LIN {X 0,Y 412.801,Z 579.645,A -85,B 0,C 180,E1 -10545.301,E2 -10545.301} C_VEL
LIN {X 0,Y 413.785,Z 567.872,A -85,B 0,C 180,E1 -10546.655,E2 -10546.655} C_VEL
LIN {X 0,Y 414.83,Z 556.165,A -85,B 0,C 180,E1 -10547.755,E2 -10547.755} C_VEL
LIN {X 0,Y 415.847,Z 543.386,A -85,B 0,C 180,E1 -10548.73,E2 -10548.73} C_VEL
LIN {X 0,Y 416.624,Z 531.359,A -85,B 0,C 180,E1 -10549.46,E2 -10549.46} C_VEL
LIN {X 0,Y 414.513,Z 516.688,A -85,B 0,C 180,E1 -10550.265,E2 -10550.265} C_VEL
LIN {X 0,Y 411.69,Z 501.521,A -85,B 0,C 180,E1 -10550.902,E2 -10550.902} C_VEL
LIN {X 0,Y 410.791,Z 496.633,A -85,B 0,C 180,E1 -10551.088,E2 -10551.088} C_VEL
LIN {X 0,Y 411.227,Z 488.281,A -85,B 0,C 180,E1 -10554.65,E2 -10554.65} C_VEL
LIN {X 0,Y 411.681,Z 480.635,A -85,B 0,C 180,E1 -10557.999,E2 -10557.999} C_VEL
LIN {X 0,Y 412.119,Z 474.429,A -85,B 0,C 180,E1 -10560.77,E2 -10560.77} C_VEL
LIN {X 0,Y 412.63,Z 468.653,A -85,B 0,C 180,E1 -10563.428,E2 -10563.428} C_VEL
LIN {X 0,Y 413.208,Z 461.279,A -85,B 0,C 180,E1 -10566.928,E2 -10566.928} C_VEL
LIN {X 0,Y 413.477,Z 457.145,A -85,B 0,C 180,E1 -10568.968,E2 -10568.968} C_VEL
LIN {X 0,Y 412.933,Z 452.303,A -85,B 0,C 180,E1 -10571.508,E2 -10571.508} C_VEL
LIN {X 0,Y 411.832,Z 446.077,A -85,B 0,C 180,E1 -10574.979,E2 -10574.979} C_VEL
LIN {X 0,Y 411.236,Z 442.884,A -85,B 0,C 180,E1 -10576.875,E2 -10576.875} C_VEL
LIN {X 0,Y 411.214,Z 442.889,A -85,B 0,C 180,E1 -10580.271,E2 -10580.271} C_VEL
LIN {X 0,Y 411.188,Z 442.891,A -85,B 0,C 180,E1 -10583.447,E2 -10583.447} C_VEL
LIN {X 0,Y 411.203,Z 442.89,A -85,B 0,C 180,E1 -10586.873,E2 -10586.873} C_VEL
LIN {X 0,Y 411.236,Z 442.886,A -85,B 0,C 180,E1 -10590.642,E2 -10590.642} C_VEL
LIN {X 0,Y 411.233,Z 442.885,A -85,B 0,C 180,E1 -10593.619,E2 -10593.619} C_VEL
LIN {X 0,Y 411.197,Z 442.892,A -85,B 0,C 180,E1 -10596.852,E2 -10596.852} C_VEL
LIN {X 0,Y 411.209,Z 442.888,A -85,B 0,C 180,E1 -10600.05,E2 -10600.05} C_VEL
LIN {X 0,Y 411.257,Z 442.883,A -85,B 0,C 180,E1 -10603.131,E2 -10603.131} C_VEL
LIN {X 0,Y 411.299,Z 442.879,A -85,B 0,C 180,E1 -10606.896,E2 -10606.896} C_VEL
LIN {X 0,Y 411.288,Z 442.878,A -85,B 0,C 180,E1 -10610.161,E2 -10610.161} C_VEL
LIN {X 0,Y 411.454,Z 442.859,A -85,B 0,C 180,E1 -10613.133,E2 -10613.133} C_VEL
LIN {X 0,Y 411.307,Z 442.876,A -85,B 0,C 180,E1 -10615.099,E2 -10615.099} C_VEL
LIN {X 0,Y 411.508,Z 442.851,A -85,B 0,C 180,E1 -10618.043,E2 -10618.043} C_VEL
LIN {X 0,Y 411.635,Z 442.834,A -85,B 0,C 180,E1 -10620,E2 -10620} C_VEL
LIN {X 0,Y 411.462,Z 442.858,A -85,B 0,C 180,E1 -10622.937,E2 -10622.937} C_VEL
LIN {X 0,Y 411.453,Z 442.858,A -85,B 0,C 180,E1 -10626.597,E2 -10626.597} C_VEL
LIN {X 0,Y 411.348,Z 442.871,A -85,B 0,C 180,E1 -10628.846,E2 -10628.846} C_VEL
LIN {X 0,Y 411.278,Z 442.88,A -85,B 0,C 180,E1 -10631.833,E2 -10631.833} C_VEL
LIN {X 0,Y 411.254,Z 442.884,A -85,B 0,C 180,E1 -10634.853,E2 -10634.853} C_VEL
LIN {X 0,Y 411.247,Z 442.883,A -85,B 0,C 180,E1 -10637.916,E2 -10637.916} C_VEL
LIN {X 0,Y 411.191,Z 442.89,A -85,B 0,C 180,E1 -10641.035,E2 -10641.035} C_VEL
LIN {X 0,Y 411.223,Z 442.888,A -85,B 0,C 180,E1 -10644.216,E2 -10644.216} C_VEL
LIN {X 0,Y 411.254,Z 442.881,A -85,B 0,C 180,E1 -10647.478,E2 -10647.478} C_VEL
LIN {X 0,Y 411.185,Z 442.89,A -85,B 0,C 180,E1 -10650.848,E2 -10650.848} C_VEL
LIN {X 0,Y 411.203,Z 442.891,A -85,B 0,C 180,E1 -10654.334,E2 -10654.334} C_VEL
LIN {X 0,Y 411.196,Z 442.892,A -85,B 0,C 180,E1 -10657.974,E2 -10657.974} C_VEL
LIN {X 0,Y 411.162,Z 442.892,A -85,B 0,C 180,E1 -10661.229,E2 -10661.229} C_VEL
LIN {X 0,Y 411.178,Z 442.892,A -85,B 0,C 180,E1 -10664.491,E2 -10664.491} C_VEL
LIN {X 0,Y 411.197,Z 442.892,A -85,B 0,C 180,E1 -10668.198,E2 -10668.198} C_VEL
LIN {X 0,Y 411.23,Z 442.885,A -85,B 0,C 180,E1 -10670.778,E2 -10670.778} C_VEL
LIN {X 0,Y 411.2,Z 442.889,A -85,B 0,C 180,E1 -10674.472,E2 -10674.472} C_VEL
LIN {X 0,Y 411.208,Z 442.887,A -85,B 0,C 180,E1 -10676.874,E2 -10676.874} C_VEL
LIN {X 0,Y 411.242,Z 442.883,A -85,B 0,C 180,E1 -10680.643,E2 -10680.643} C_VEL
LIN {X 0,Y 411.24,Z 442.887,A -85,B 0,C 180,E1 -10683.62,E2 -10683.62} C_VEL
LIN {X 0,Y 411.206,Z 442.887,A -85,B 0,C 180,E1 -10686.853,E2 -10686.853} C_VEL
LIN {X 0,Y 411.218,Z 442.889,A -85,B 0,C 180,E1 -10690.051,E2 -10690.051} C_VEL
LIN {X 0,Y 411.266,Z 442.881,A -85,B 0,C 180,E1 -10693.132,E2 -10693.132} C_VEL
LIN {X 0,Y 411.309,Z 442.874,A -85,B 0,C 180,E1 -10696.896,E2 -10696.896} C_VEL
LIN {X 0,Y 411.296,Z 442.877,A -85,B 0,C 180,E1 -10700.162,E2 -10700.162} C_VEL
LIN {X 0,Y 411.427,Z 442.863,A -85,B 0,C 180,E1 -10703.133,E2 -10703.133} C_VEL
LIN {X 0,Y 411.31,Z 442.876,A -85,B 0,C 180,E1 -10705.099,E2 -10705.099} C_VEL
LIN {X 0,Y 411.518,Z 442.85,A -85,B 0,C 180,E1 -10708.043,E2 -10708.043} C_VEL
LIN {X 0,Y 411.644,Z 442.833,A -85,B 0,C 180,E1 -10710,E2 -10710} C_VEL
LIN {X 0,Y 411.462,Z 442.858,A -85,B 0,C 180,E1 -10712.937,E2 -10712.937} C_VEL
LIN {X 0,Y 411.475,Z 442.855,A -85,B 0,C 180,E1 -10715.882,E2 -10715.882} C_VEL
LIN {X 0,Y 411.355,Z 442.87,A -85,B 0,C 180,E1 -10718.845,E2 -10718.845} C_VEL
LIN {X 0,Y 411.288,Z 442.879,A -85,B 0,C 180,E1 -10721.832,E2 -10721.832} C_VEL
LIN {X 0,Y 411.263,Z 442.883,A -85,B 0,C 180,E1 -10724.852,E2 -10724.852} C_VEL
LIN {X 0,Y 411.243,Z 442.881,A -85,B 0,C 180,E1 -10727.596,E2 -10727.596} C_VEL
LIN {X 0,Y 410.583,Z 442.965,A -85,B 0,C 180,E1 -10728.414,E2 -10728.414} C_VEL
LIN {X 0,Y 407.695,Z 443.326,A -85,B 0,C 180,E1 -10729.742,E2 -10729.742} C_VEL
LIN {X 0,Y 405.25,Z 443.632,A -85,B 0,C 180,E1 -10730.814,E2 -10730.814} C_VEL
LIN {X 0,Y 404.215,Z 443.76,A -85,B 0,C 180,E1 -10731.644,E2 -10731.644} C_VEL
LIN {X 0,Y 404.139,Z 443.767,A -85,B 0,C 180,E1 -10731.926,E2 -10731.926} C_VEL
LIN {X 0,Y 404.218,Z 443.761,A -85,B 0,C 180,E1 -10735.296,E2 -10735.296} C_VEL
LIN {X 0,Y 404.197,Z 443.76,A -85,B 0,C 180,E1 -10737.999,E2 -10737.999} C_VEL
LIN {X 0,Y 404.138,Z 443.768,A -85,B 0,C 180,E1 -10741.557,E2 -10741.557} C_VEL
LIN {X 0,Y 404.105,Z 443.772,A -85,B 0,C 180,E1 -10743.815,E2 -10743.815} C_VEL
LIN {X 0,Y 403.874,Z 443.805,A -85,B 0,C 180,E1 -10746.825,E2 -10746.825} C_VEL
LIN {X 0,Y 403.436,Z 443.861,A -85,B 0,C 180,E1 -10750.131,E2 -10750.131} C_VEL
LIN {X 0,Y 403.357,Z 444.539,A -85,B 0,C 180,E1 -10751.476,E2 -10751.476} C_VEL
LIN {X 0,Y 403.264,Z 447.096,A -85,B 0,C 180,E1 -10754.394,E2 -10754.394} C_VEL
LIN {X 0,Y 403.237,Z 449.596,A -85,B 0,C 180,E1 -10757.177,E2 -10757.177} C_VEL
LIN {X 0,Y 403.147,Z 452.843,A -85,B 0,C 180,E1 -10760.723,E2 -10760.723} C_VEL
LIN {X 0,Y 407.346,Z 467.682,A -85,B 0,C 180,E1 -10761.418,E2 -10761.418} C_VEL
LIN {X 0,Y 410.494,Z 480.117,A -85,B 0,C 180,E1 -10762.156,E2 -10762.156} C_VEL
LIN {X 0,Y 409.792,Z 493.988,A -85,B 0,C 180,E1 -10762.977,E2 -10762.977} C_VEL
LIN {X 0,Y 408.853,Z 507.194,A -85,B 0,C 180,E1 -10763.977,E2 -10763.977} C_VEL
LIN {X 0,Y 407.914,Z 518.652,A -85,B 0,C 180,E1 -10765.049,E2 -10765.049} C_VEL
LIN {X 0,Y 406.818,Z 530.774,A -85,B 0,C 180,E1 -10766.439,E2 -10766.439} C_VEL
LIN {X 0,Y 405.964,Z 540.883,A -85,B 0,C 180,E1 -10767.852,E2 -10767.852} C_VEL
LIN {X 0,Y 405.008,Z 550.623,A -85,B 0,C 180,E1 -10769.498,E2 -10769.498} C_VEL
LIN {X 0,Y 404.378,Z 558.657,A -85,B 0,C 180,E1 -10771.165,E2 -10771.165} C_VEL
LIN {X 0,Y 403.791,Z 566.103,A -85,B 0,C 180,E1 -10773.093,E2 -10773.093} C_VEL
LIN {X 0,Y 403.401,Z 571.667,A -85,B 0,C 180,E1 -10774.948,E2 -10774.948} C_VEL
LIN {X 0,Y 403.096,Z 576.05,A -85,B 0,C 180,E1 -10776.903,E2 -10776.903} C_VEL
LIN {X 0,Y 402.928,Z 578.626,A -85,B 0,C 180,E1 -10778.513,E2 -10778.513} C_VEL
LIN {X 0,Y 402.891,Z 580.598,A -85,B 0,C 180,E1 -10780.644,E2 -10780.644} C_VEL
LIN {X 0,Y 402.812,Z 581.067,A -85,B 0,C 180,E1 -10782.746,E2 -10782.746} C_VEL
LIN {X 0,Y 402.892,Z 580.745,A -85,B 0,C 180,E1 -10783.793,E2 -10783.793} C_VEL
LIN {X 0,Y 402.994,Z 579.036,A -85,B 0,C 180,E1 -10785.868,E2 -10785.868} C_VEL
LIN {X 0,Y 403.289,Z 575.854,A -85,B 0,C 180,E1 -10787.929,E2 -10787.929} C_VEL
LIN {X 0,Y 403.699,Z 571.129,A -85,B 0,C 180,E1 -10789.974,E2 -10789.974} C_VEL
LIN {X 0,Y 404.133,Z 566.55,A -85,B 0,C 180,E1 -10791.499,E2 -10791.499} C_VEL
LIN {X 0,Y 404.794,Z 559.874,A -85,B 0,C 180,E1 -10793.27,E2 -10793.27} C_VEL
LIN {X 0,Y 405.692,Z 551.582,A -85,B 0,C 180,E1 -10795.031,E2 -10795.031} C_VEL
LIN {X 0,Y 406.521,Z 543.028,A -85,B 0,C 180,E1 -10796.531,E2 -10796.531} C_VEL
LIN {X 0,Y 407.677,Z 532.688,A -85,B 0,C 180,E1 -10798.024,E2 -10798.024} C_VEL
LIN {X 0,Y 408.851,Z 521.23,A -85,B 0,C 180,E1 -10799.384,E2 -10799.384} C_VEL
LIN {X 0,Y 409.933,Z 509.849,A -85,B 0,C 180,E1 -10800.491,E2 -10800.491} C_VEL
LIN {X 0,Y 410.984,Z 497.505,A -85,B 0,C 180,E1 -10801.47,E2 -10801.47} C_VEL
LIN {X 0,Y 411.945,Z 484.382,A -85,B 0,C 180,E1 -10802.291,E2 -10802.291} C_VEL
LIN {X 0,Y 411.781,Z 481.336,A -85,B 0,C 180,E1 -10802.475,E2 -10802.475} C_VEL
LIN {X 0,Y 408.191,Z 469.01,A -85,B 0,C 180,E1 -10803.332,E2 -10803.332} C_VEL
LIN {X 0,Y 403.763,Z 456.429,A -85,B 0,C 180,E1 -10804.117,E2 -10804.117} C_VEL
LIN {X 0,Y 403.9,Z 455.086,A -85,B 0,C 180,E1 -10805.993,E2 -10805.993} C_VEL
LIN {X 0,Y 404.002,Z 453.036,A -85,B 0,C 180,E1 -10809.007,E2 -10809.007} C_VEL
LIN {X 0,Y 404.199,Z 450.477,A -85,B 0,C 180,E1 -10813.064,E2 -10813.064} C_VEL
LIN {X 0,Y 404.4,Z 448.23,A -85,B 0,C 180,E1 -10817.095,E2 -10817.095} C_VEL
LIN {X 0,Y 404.491,Z 446.675,A -85,B 0,C 180,E1 -10820.334,E2 -10820.334} C_VEL
LIN {X 0,Y 404.408,Z 445.473,A -85,B 0,C 180,E1 -10823.56,E2 -10823.56} C_VEL
LIN {X 0,Y 404.338,Z 444.649,A -85,B 0,C 180,E1 -10826.867,E2 -10826.867} C_VEL
LIN {X 0,Y 404.254,Z 444.334,A -85,B 0,C 180,E1 -10830.276,E2 -10830.276} C_VEL
LIN {X 0,Y 404.31,Z 444.687,A -85,B 0,C 180,E1 -10833.796,E2 -10833.796} C_VEL
LIN {X 0,Y 404.476,Z 445.696,A -85,B 0,C 180,E1 -10836.94,E2 -10836.94} C_VEL
LIN {X 0,Y 404.854,Z 447.496,A -85,B 0,C 180,E1 -10840.2,E2 -10840.2} C_VEL
LIN {X 0,Y 405.277,Z 449.926,A -85,B 0,C 180,E1 -10843.254,E2 -10843.254} C_VEL
LIN {X 0,Y 405.875,Z 453.507,A -85,B 0,C 180,E1 -10846.657,E2 -10846.657} C_VEL
LIN {X 0,Y 406.437,Z 457.209,A -85,B 0,C 180,E1 -10849.538,E2 -10849.538} C_VEL
LIN {X 0,Y 406.531,Z 460.16,A -85,B 0,C 180,E1 -10851.512,E2 -10851.512} C_VEL
LIN {X 0,Y 406,Z 464.25,A -85,B 0,C 180,E1 -10853.946,E2 -10853.946} C_VEL
LIN {X 0,Y 405.372,Z 469.698,A -85,B 0,C 180,E1 -10856.899,E2 -10856.899} C_VEL
LIN {X 0,Y 404.824,Z 476.312,A -85,B 0,C 180,E1 -10860.231,E2 -10860.231} C_VEL
LIN {X 0,Y 404.208,Z 483.672,A -85,B 0,C 180,E1 -10863.681,E2 -10863.681} C_VEL
LIN {X 0,Y 403.747,Z 492.25,A -85,B 0,C 180,E1 -10867.484,E2 -10867.484} C_VEL
LIN {X 0,Y 403.739,Z 493.024,A -85,B 0,C 180,E1 -10867.818,E2 -10867.818} C_VEL
LIN {X 0,Y 407.633,Z 510.63,A -85,B 0,C 180,E1 -10868.708,E2 -10868.708} C_VEL
LIN {X 0,Y 409.371,Z 523.324,A -85,B 0,C 180,E1 -10869.428,E2 -10869.428} C_VEL
LIN {X 0,Y 410.314,Z 533.68,A -85,B 0,C 180,E1 -10870.098,E2 -10870.098} C_VEL
LIN {X 0,Y 409.062,Z 547.719,A -85,B 0,C 180,E1 -10871.078,E2 -10871.078} C_VEL
LIN {X 0,Y 407.899,Z 560.436,A -85,B 0,C 180,E1 -10872.192,E2 -10872.192} C_VEL
LIN {X 0,Y 406.715,Z 572.083,A -85,B 0,C 180,E1 -10873.434,E2 -10873.434} C_VEL
LIN {X 0,Y 405.589,Z 583.695,A -85,B 0,C 180,E1 -10874.935,E2 -10874.935} C_VEL
LIN {X 0,Y 404.658,Z 593.952,A -85,B 0,C 180,E1 -10876.555,E2 -10876.555} C_VEL
LIN {X 0,Y 404.026,Z 602.53,A -85,B 0,C 180,E1 -10878.206,E2 -10878.206} C_VEL
LIN {X 0,Y 403.45,Z 610.025,A -85,B 0,C 180,E1 -10879.968,E2 -10879.968} C_VEL
LIN {X 0,Y 403.169,Z 615.304,A -85,B 0,C 180,E1 -10881.479,E2 -10881.479} C_VEL
LIN {X 0,Y 403.068,Z 619.556,A -85,B 0,C 180,E1 -10882.989,E2 -10882.989} C_VEL
LIN {X 0,Y 402.944,Z 623.879,A -85,B 0,C 180,E1 -10884.997,E2 -10884.997} C_VEL
LIN {X 0,Y 402.948,Z 626.705,A -85,B 0,C 180,E1 -10887.001,E2 -10887.001} C_VEL
LIN {X 0,Y 402.981,Z 627.576,A -85,B 0,C 180,E1 -10888.001,E2 -10888.001} C_VEL
LIN {X 0,Y 402.95,Z 628.259,A -85,B 0,C 180,E1 -10890,E2 -10890} C_VEL
LIN {X 0,Y 402.981,Z 627.549,A -85,B 0,C 180,E1 -10891.999,E2 -10891.999} C_VEL
LIN {X 0,Y 402.877,Z 625.421,A -85,B 0,C 180,E1 -10894.001,E2 -10894.001} C_VEL
LIN {X 0,Y 402.955,Z 623.822,A -85,B 0,C 180,E1 -10895.003,E2 -10895.003} C_VEL
LIN {X 0,Y 403.064,Z 619.474,A -85,B 0,C 180,E1 -10897.011,E2 -10897.011} C_VEL
LIN {X 0,Y 403.27,Z 613.496,A -85,B 0,C 180,E1 -10899.024,E2 -10899.024} C_VEL
LIN {X 0,Y 403.653,Z 606.738,A -85,B 0,C 180,E1 -10900.787,E2 -10900.787} C_VEL
LIN {X 0,Y 404.335,Z 598.312,A -85,B 0,C 180,E1 -10902.549,E2 -10902.549} C_VEL
LIN {X 0,Y 404.942,Z 589.515,A -85,B 0,C 180,E1 -10904.062,E2 -10904.062} C_VEL
LIN {X 0,Y 405.88,Z 578.894,A -85,B 0,C 180,E1 -10905.568,E2 -10905.568} C_VEL
LIN {X 0,Y 406.897,Z 567.057,A -85,B 0,C 180,E1 -10906.946,E2 -10906.946} C_VEL
LIN {X 0,Y 407.993,Z 555.275,A -85,B 0,C 180,E1 -10908.063,E2 -10908.063} C_VEL
LIN {X 0,Y 409.075,Z 542.402,A -85,B 0,C 180,E1 -10909.051,E2 -10909.051} C_VEL
LIN {X 0,Y 409.624,Z 531.3,A -85,B 0,C 180,E1 -10909.741,E2 -10909.741} C_VEL
LIN {X 0,Y 407.503,Z 516.685,A -85,B 0,C 180,E1 -10910.568,E2 -10910.568} C_VEL
LIN {X 0,Y 404.728,Z 501.456,A -85,B 0,C 180,E1 -10911.228,E2 -10911.228} C_VEL
LIN {X 0,Y 403.718,Z 496.266,A -85,B 0,C 180,E1 -10911.442,E2 -10911.442} C_VEL
LIN {X 0,Y 404.152,Z 488.877,A -85,B 0,C 180,E1 -10914.667,E2 -10914.667} C_VEL
LIN {X 0,Y 404.619,Z 481.458,A -85,B 0,C 180,E1 -10917.967,E2 -10917.967} C_VEL
LIN {X 0,Y 405.087,Z 475.295,A -85,B 0,C 180,E1 -10920.784,E2 -10920.784} C_VEL
LIN {X 0,Y 405.626,Z 469.009,A -85,B 0,C 180,E1 -10923.73,E2 -10923.73} C_VEL
LIN {X 0,Y 406.249,Z 461.72,A -85,B 0,C 180,E1 -10927.27,E2 -10927.27} C_VEL
LIN {X 0,Y 406.486,Z 458.432,A -85,B 0,C 180,E1 -10928.919,E2 -10928.919} C_VEL
LIN {X 0,Y 406.082,Z 454.284,A -85,B 0,C 180,E1 -10931.121,E2 -10931.121} C_VEL
LIN {X 0,Y 404.965,Z 448.024,A -85,B 0,C 180,E1 -10934.64,E2 -10934.64} C_VEL
LIN {X 0,Y 404.216,Z 443.758,A -85,B 0,C 180,E1 -10937.306,E2 -10937.306} C_VEL
LIN {X 0,Y 404.165,Z 443.766,A -85,B 0,C 180,E1 -10939.955,E2 -10939.955} C_VEL
LIN {X 0,Y 404.132,Z 443.772,A -85,B 0,C 180,E1 -10943.125,E2 -10943.125} C_VEL
LIN {X 0,Y 404.14,Z 443.768,A -85,B 0,C 180,E1 -10946.187,E2 -10946.187} C_VEL
LIN {X 0,Y 404.151,Z 443.767,A -85,B 0,C 180,E1 -10949.715,E2 -10949.715} C_VEL
LIN {X 0,Y 404.19,Z 443.764,A -85,B 0,C 180,E1 -10953.123,E2 -10953.123} C_VEL
LIN {X 0,Y 404.172,Z 443.766,A -85,B 0,C 180,E1 -10955.334,E2 -10955.334} C_VEL
LIN {X 0,Y 404.133,Z 443.771,A -85,B 0,C 180,E1 -10958.58,E2 -10958.58} C_VEL
LIN {X 0,Y 404.204,Z 443.758,A -85,B 0,C 180,E1 -10961.762,E2 -10961.762} C_VEL
LIN {X 0,Y 404.2,Z 443.764,A -85,B 0,C 180,E1 -10964.882,E2 -10964.882} C_VEL
LIN {X 0,Y 404.251,Z 443.754,A -85,B 0,C 180,E1 -10967.959,E2 -10967.959} C_VEL
LIN {X 0,Y 404.427,Z 443.733,A -85,B 0,C 180,E1 -10972.1,E2 -10972.1} C_VEL
LIN {X 0,Y 404.418,Z 443.734,A -85,B 0,C 180,E1 -10974.015,E2 -10974.015} C_VEL
LIN {X 0,Y 404.477,Z 443.727,A -85,B 0,C 180,E1 -10978.009,E2 -10978.009} C_VEL
LIN {X 0,Y 404.605,Z 443.71,A -85,B 0,C 180,E1 -10980,E2 -10980} C_VEL
LIN {X 0,Y 404.419,Z 443.735,A -85,B 0,C 180,E1 -10982.989,E2 -10982.989} C_VEL
LIN {X 0,Y 404.403,Z 443.735,A -85,B 0,C 180,E1 -10986.595,E2 -10986.595} C_VEL
LIN {X 0,Y 404.285,Z 443.75,A -85,B 0,C 180,E1 -10989.001,E2 -10989.001} C_VEL
LIN {X 0,Y 404.25,Z 443.756,A -85,B 0,C 180,E1 -10992.042,E2 -10992.042} C_VEL
LIN {X 0,Y 404.2,Z 443.761,A -85,B 0,C 180,E1 -10995.118,E2 -10995.118} C_VEL
LIN {X 0,Y 404.205,Z 443.763,A -85,B 0,C 180,E1 -10998.239,E2 -10998.239} C_VEL
LIN {X 0,Y 404.134,Z 443.768,A -85,B 0,C 180,E1 -11001.42,E2 -11001.42} C_VEL
LIN {X 0,Y 404.173,Z 443.766,A -85,B 0,C 180,E1 -11004.666,E2 -11004.666} C_VEL
LIN {X 0,Y 404.191,Z 443.765,A -85,B 0,C 180,E1 -11008,E2 -11008} C_VEL
LIN {X 0,Y 404.135,Z 443.768,A -85,B 0,C 180,E1 -11011.559,E2 -11011.559} C_VEL
LIN {X 0,Y 404.182,Z 443.762,A -85,B 0,C 180,E1 -11015.017,E2 -11015.017} C_VEL
LIN {X 0,Y 404.153,Z 443.767,A -85,B 0,C 180,E1 -11018.757,E2 -11018.757} C_VEL
LIN {X 0,Y 404.122,Z 443.771,A -85,B 0,C 180,E1 -11021.601,E2 -11021.601} C_VEL
LIN {X 0,Y 404.147,Z 443.767,A -85,B 0,C 180,E1 -11024.523,E2 -11024.523} C_VEL
LIN {X 0,Y 404.17,Z 443.765,A -85,B 0,C 180,E1 -11027.301,E2 -11027.301} C_VEL
LIN {X 0,Y 404.168,Z 443.768,A -85,B 0,C 180,E1 -11029.956,E2 -11029.956} C_VEL
LIN {X 0,Y 404.141,Z 443.768,A -85,B 0,C 180,E1 -11033.125,E2 -11033.125} C_VEL
LIN {X 0,Y 404.146,Z 443.77,A -85,B 0,C 180,E1 -11036.189,E2 -11036.189} C_VEL
LIN {X 0,Y 404.155,Z 443.769,A -85,B 0,C 180,E1 -11039.716,E2 -11039.716} C_VEL
LIN {X 0,Y 404.197,Z 443.76,A -85,B 0,C 180,E1 -11043.124,E2 -11043.124} C_VEL
LIN {X 0,Y 404.18,Z 443.765,A -85,B 0,C 180,E1 -11045.335,E2 -11045.335} C_VEL
LIN {X 0,Y 404.141,Z 443.767,A -85,B 0,C 180,E1 -11048.581,E2 -11048.581} C_VEL
LIN {X 0,Y 404.213,Z 443.762,A -85,B 0,C 180,E1 -11051.762,E2 -11051.762} C_VEL
LIN {X 0,Y 404.21,Z 443.76,A -85,B 0,C 180,E1 -11054.882,E2 -11054.882} C_VEL
LIN {X 0,Y 404.26,Z 443.755,A -85,B 0,C 180,E1 -11057.959,E2 -11057.959} C_VEL
LIN {X 0,Y 404.292,Z 443.749,A -85,B 0,C 180,E1 -11060.999,E2 -11060.999} C_VEL
LIN {X 0,Y 404.397,Z 443.737,A -85,B 0,C 180,E1 -11064.015,E2 -11064.015} C_VEL
LIN {X 0,Y 404.487,Z 443.726,A -85,B 0,C 180,E1 -11068.009,E2 -11068.009} C_VEL
LIN {X 0,Y 404.614,Z 443.708,A -85,B 0,C 180,E1 -11070,E2 -11070} C_VEL
LIN {X 0,Y 404.42,Z 443.735,A -85,B 0,C 180,E1 -11072.988,E2 -11072.988} C_VEL
LIN {X 0,Y 404.422,Z 443.733,A -85,B 0,C 180,E1 -11075.985,E2 -11075.985} C_VEL
LIN {X 0,Y 404.292,Z 443.751,A -85,B 0,C 180,E1 -11079.001,E2 -11079.001} C_VEL
LIN {X 0,Y 404.26,Z 443.753,A -85,B 0,C 180,E1 -11082.041,E2 -11082.041} C_VEL
LIN {X 0,Y 404.21,Z 443.762,A -85,B 0,C 180,E1 -11085.118,E2 -11085.118} C_VEL
LIN {X 0,Y 404.213,Z 443.757,A -85,B 0,C 180,E1 -11088.238,E2 -11088.238} C_VEL
LIN {X 0,Y 404.141,Z 443.77,A -85,B 0,C 180,E1 -11091.419,E2 -11091.419} C_VEL
LIN {X 0,Y 404.139,Z 443.767,A -85,B 0,C 180,E1 -11091.926,E2 -11091.926} C_VEL
LIN {X 0,Y 403.497,Z 443.851,A -85,B 0,C 180,E1 -11092.757,E2 -11092.757} C_VEL
LIN {X 0,Y 400.664,Z 444.203,A -85,B 0,C 180,E1 -11094.109,E2 -11094.109} C_VEL
LIN {X 0,Y 398.254,Z 444.504,A -85,B 0,C 180,E1 -11095.201,E2 -11095.201} C_VEL
LIN {X 0,Y 397.219,Z 444.631,A -85,B 0,C 180,E1 -11096.045,E2 -11096.045} C_VEL
LIN {X 0,Y 397.136,Z 444.639,A -85,B 0,C 180,E1 -11096.331,E2 -11096.331} C_VEL
LIN {X 0,Y 397.124,Z 444.643,A -85,B 0,C 180,E1 -11098.543,E2 -11098.543} C_VEL
LIN {X 0,Y 397.075,Z 444.646,A -85,B 0,C 180,E1 -11102.071,E2 -11102.071} C_VEL
LIN {X 0,Y 397.018,Z 444.657,A -85,B 0,C 180,E1 -11104.503,E2 -11104.503} C_VEL
LIN {X 0,Y 396.761,Z 444.69,A -85,B 0,C 180,E1 -11107.145,E2 -11107.145} C_VEL
LIN {X 0,Y 396.382,Z 444.739,A -85,B 0,C 180,E1 -11110.323,E2 -11110.323} C_VEL
LIN {X 0,Y 396.293,Z 444.863,A -85,B 0,C 180,E1 -11111.008,E2 -11111.008} C_VEL
LIN {X 0,Y 396.224,Z 447.255,A -85,B 0,C 180,E1 -11113.769,E2 -11113.769} C_VEL
LIN {X 0,Y 396.143,Z 450.68,A -85,B 0,C 180,E1 -11117.611,E2 -11117.611} C_VEL
LIN {X 0,Y 396.086,Z 453.187,A -85,B 0,C 180,E1 -11120.365,E2 -11120.365} C_VEL
LIN {X 0,Y 400.798,Z 469.92,A -85,B 0,C 180,E1 -11121.197,E2 -11121.197} C_VEL
LIN {X 0,Y 403.757,Z 481.786,A -85,B 0,C 180,E1 -11121.929,E2 -11121.929} C_VEL
LIN {X 0,Y 402.919,Z 495.445,A -85,B 0,C 180,E1 -11122.768,E2 -11122.768} C_VEL
LIN {X 0,Y 401.902,Z 508.896,A -85,B 0,C 180,E1 -11123.83,E2 -11123.83} C_VEL
LIN {X 0,Y 400.83,Z 521.361,A -85,B 0,C 180,E1 -11125.054,E2 -11125.054} C_VEL
LIN {X 0,Y 399.823,Z 532.406,A -85,B 0,C 180,E1 -11126.378,E2 -11126.378} C_VEL
LIN {X 0,Y 398.93,Z 542.406,A -85,B 0,C 180,E1 -11127.828,E2 -11127.828} C_VEL
LIN {X 0,Y 397.983,Z 551.538,A -85,B 0,C 180,E1 -11129.422,E2 -11129.422} C_VEL
LIN {X 0,Y 397.305,Z 559.75,A -85,B 0,C 180,E1 -11131.182,E2 -11131.182} C_VEL
LIN {X 0,Y 396.717,Z 567.029,A -85,B 0,C 180,E1 -11133.144,E2 -11133.144} C_VEL
LIN {X 0,Y 396.359,Z 571.943,A -85,B 0,C 180,E1 -11134.814,E2 -11134.814} C_VEL
LIN {X 0,Y 396.093,Z 575.755,A -85,B 0,C 180,E1 -11136.47,E2 -11136.47} C_VEL
LIN {X 0,Y 395.882,Z 578.512,A -85,B 0,C 180,E1 -11138.111,E2 -11138.111} C_VEL
LIN {X 0,Y 395.811,Z 580.814,A -85,B 0,C 180,E1 -11140.283,E2 -11140.283} C_VEL
LIN {X 0,Y 395.734,Z 581.534,A -85,B 0,C 180,E1 -11142.427,E2 -11142.427} C_VEL
LIN {X 0,Y 395.826,Z 580.778,A -85,B 0,C 180,E1 -11144.554,E2 -11144.554} C_VEL
LIN {X 0,Y 396.013,Z 578.587,A -85,B 0,C 180,E1 -11146.661,E2 -11146.661} C_VEL
LIN {X 0,Y 396.397,Z 574.932,A -85,B 0,C 180,E1 -11148.753,E2 -11148.753} C_VEL
LIN {X 0,Y 396.737,Z 571.155,A -85,B 0,C 180,E1 -11150.311,E2 -11150.311} C_VEL
LIN {X 0,Y 397.386,Z 564.756,A -85,B 0,C 180,E1 -11152.356,E2 -11152.356} C_VEL
LIN {X 0,Y 398.207,Z 557.496,A -85,B 0,C 180,E1 -11154.175,E2 -11154.175} C_VEL
LIN {X 0,Y 399.198,Z 548.587,A -85,B 0,C 180,E1 -11155.962,E2 -11155.962} C_VEL
LIN {X 0,Y 400.253,Z 539.312,A -85,B 0,C 180,E1 -11157.484,E2 -11157.484} C_VEL
LIN {X 0,Y 401.508,Z 528.079,A -85,B 0,C 180,E1 -11158.997,E2 -11158.997} C_VEL
LIN {X 0,Y 402.686,Z 516.727,A -85,B 0,C 180,E1 -11160.25,E2 -11160.25} C_VEL
LIN {X 0,Y 403.878,Z 504.362,A -85,B 0,C 180,E1 -11161.371,E2 -11161.371} C_VEL
LIN {X 0,Y 405.002,Z 491.224,A -85,B 0,C 180,E1 -11162.318,E2 -11162.318} C_VEL
LIN {X 0,Y 405.512,Z 484.018,A -85,B 0,C 180,E1 -11162.746,E2 -11162.746} C_VEL
LIN {X 0,Y 402.095,Z 471.959,A -85,B 0,C 180,E1 -11163.633,E2 -11163.633} C_VEL
LIN {X 0,Y 397.322,Z 458.967,A -85,B 0,C 180,E1 -11164.518,E2 -11164.518} C_VEL
LIN {X 0,Y 396.823,Z 457.011,A -85,B 0,C 180,E1 -11164.635,E2 -11164.635} C_VEL
LIN {X 0,Y 396.975,Z 454.625,A -85,B 0,C 180,E1 -11168.142,E2 -11168.142} C_VEL
LIN {X 0,Y 397.05,Z 452.67,A -85,B 0,C 180,E1 -11171.227,E2 -11171.227} C_VEL
LIN {X 0,Y 397.193,Z 450.858,A -85,B 0,C 180,E1 -11174.342,E2 -11174.342} C_VEL
LIN {X 0,Y 397.409,Z 449.208,A -85,B 0,C 180,E1 -11177.496,E2 -11177.496} C_VEL
LIN {X 0,Y 397.477,Z 447.778,A -85,B 0,C 180,E1 -11180.709,E2 -11180.709} C_VEL
LIN {X 0,Y 397.41,Z 446.679,A -85,B 0,C 180,E1 -11184,E2 -11184} C_VEL
LIN {X 0,Y 397.389,Z 445.966,A -85,B 0,C 180,E1 -11187.375,E2 -11187.375} C_VEL
LIN {X 0,Y 397.301,Z 445.823,A -85,B 0,C 180,E1 -11190.863,E2 -11190.863} C_VEL
LIN {X 0,Y 397.398,Z 446.37,A -85,B 0,C 180,E1 -11194.466,E2 -11194.466} C_VEL
LIN {X 0,Y 397.673,Z 447.853,A -85,B 0,C 180,E1 -11198.21,E2 -11198.21} C_VEL
LIN {X 0,Y 397.995,Z 449.458,A -85,B 0,C 180,E1 -11200.796,E2 -11200.796} C_VEL
LIN {X 0,Y 398.403,Z 451.845,A -85,B 0,C 180,E1 -11203.677,E2 -11203.677} C_VEL
LIN {X 0,Y 398.931,Z 454.897,A -85,B 0,C 180,E1 -11206.603,E2 -11206.603} C_VEL
LIN {X 0,Y 399.464,Z 458.385,A -85,B 0,C 180,E1 -11209.387,E2 -11209.387} C_VEL
LIN {X 0,Y 399.543,Z 460.286,A -85,B 0,C 180,E1 -11210.711,E2 -11210.711} C_VEL
LIN {X 0,Y 399.201,Z 464.294,A -85,B 0,C 180,E1 -11213.233,E2 -11213.233} C_VEL
LIN {X 0,Y 398.355,Z 470.713,A -85,B 0,C 180,E1 -11216.845,E2 -11216.845} C_VEL
LIN {X 0,Y 397.76,Z 477.543,A -85,B 0,C 180,E1 -11220.349,E2 -11220.349} C_VEL
LIN {X 0,Y 397.159,Z 484.639,A -85,B 0,C 180,E1 -11223.744,E2 -11223.744} C_VEL
LIN {X 0,Y 396.702,Z 492.515,A -85,B 0,C 180,E1 -11227.324,E2 -11227.324} C_VEL
LIN {X 0,Y 400.543,Z 508.904,A -85,B 0,C 180,E1 -11228.172,E2 -11228.172} C_VEL
LIN {X 0,Y 402.494,Z 521.599,A -85,B 0,C 180,E1 -11228.919,E2 -11228.919} C_VEL
LIN {X 0,Y 403.646,Z 533.983,A -85,B 0,C 180,E1 -11229.755,E2 -11229.755} C_VEL
LIN {X 0,Y 402.357,Z 547.67,A -85,B 0,C 180,E1 -11230.736,E2 -11230.736} C_VEL
LIN {X 0,Y 401.134,Z 560.44,A -85,B 0,C 180,E1 -11231.882,E2 -11231.882} C_VEL
LIN {X 0,Y 399.876,Z 572.007,A -85,B 0,C 180,E1 -11233.143,E2 -11233.143} C_VEL
LIN {X 0,Y 398.689,Z 583.519,A -85,B 0,C 180,E1 -11234.668,E2 -11234.668} C_VEL
LIN {X 0,Y 397.802,Z 592.833,A -85,B 0,C 180,E1 -11236.164,E2 -11236.164} C_VEL
LIN {X 0,Y 397.063,Z 601.041,A -85,B 0,C 180,E1 -11237.737,E2 -11237.737} C_VEL
LIN {X 0,Y 396.551,Z 607.729,A -85,B 0,C 180,E1 -11239.276,E2 -11239.276} C_VEL
LIN {X 0,Y 396.206,Z 613.297,A -85,B 0,C 180,E1 -11240.814,E2 -11240.814} C_VEL
LIN {X 0,Y 395.985,Z 619.202,A -85,B 0,C 180,E1 -11242.863,E2 -11242.863} C_VEL
LIN {X 0,Y 395.86,Z 623.502,A -85,B 0,C 180,E1 -11244.907,E2 -11244.907} C_VEL
LIN {X 0,Y 395.849,Z 626.3,A -85,B 0,C 180,E1 -11246.947,E2 -11246.947} C_VEL
LIN {X 0,Y 395.91,Z 627.163,A -85,B 0,C 180,E1 -11247.965,E2 -11247.965} C_VEL
LIN {X 0,Y 395.872,Z 627.831,A -85,B 0,C 180,E1 -11250,E2 -11250} C_VEL
LIN {X 0,Y 395.91,Z 627.103,A -85,B 0,C 180,E1 -11252.035,E2 -11252.035} C_VEL
LIN {X 0,Y 395.799,Z 624.952,A -85,B 0,C 180,E1 -11254.073,E2 -11254.073} C_VEL
LIN {X 0,Y 395.908,Z 621.346,A -85,B 0,C 180,E1 -11256.114,E2 -11256.114} C_VEL
LIN {X 0,Y 395.994,Z 617.614,A -85,B 0,C 180,E1 -11257.649,E2 -11257.649} C_VEL
LIN {X 0,Y 396.207,Z 612.948,A -85,B 0,C 180,E1 -11259.186,E2 -11259.186} C_VEL
LIN {X 0,Y 396.64,Z 606.145,A -85,B 0,C 180,E1 -11260.98,E2 -11260.98} C_VEL
LIN {X 0,Y 397.347,Z 597.667,A -85,B 0,C 180,E1 -11262.773,E2 -11262.773} C_VEL
LIN {X 0,Y 397.984,Z 588.82,A -85,B 0,C 180,E1 -11264.313,E2 -11264.313} C_VEL
LIN {X 0,Y 398.972,Z 578.145,A -85,B 0,C 180,E1 -11265.845,E2 -11265.845} C_VEL
LIN {X 0,Y 400.068,Z 566.248,A -85,B 0,C 180,E1 -11267.244,E2 -11267.244} C_VEL
LIN {X 0,Y 401.184,Z 554.388,A -85,B 0,C 180,E1 -11268.38,E2 -11268.38} C_VEL
LIN {X 0,Y 402.276,Z 541.378,A -85,B 0,C 180,E1 -11269.386,E2 -11269.386} C_VEL
LIN {X 0,Y 402.77,Z 532.349,A -85,B 0,C 180,E1 -11269.959,E2 -11269.959} C_VEL
LIN {X 0,Y 400.786,Z 518.378,A -85,B 0,C 180,E1 -11270.787,E2 -11270.787} C_VEL
LIN {X 0,Y 398.144,Z 503.438,A -85,B 0,C 180,E1 -11271.479,E2 -11271.479} C_VEL
LIN {X 0,Y 396.663,Z 495.998,A -85,B 0,C 180,E1 -11271.757,E2 -11271.757} C_VEL
LIN {X 0,Y 397.123,Z 488.433,A -85,B 0,C 180,E1 -11275.133,E2 -11275.133} C_VEL
LIN {X 0,Y 397.535,Z 482.407,A -85,B 0,C 180,E1 -11277.878,E2 -11277.878} C_VEL
LIN {X 0,Y 398.13,Z 474.894,A -85,B 0,C 180,E1 -11281.382,E2 -11281.382} C_VEL
LIN {X 0,Y 398.7,Z 468.75,A -85,B 0,C 180,E1 -11284.337,E2 -11284.337} C_VEL
LIN {X 0,Y 399.385,Z 461.347,A -85,B 0,C 180,E1 -11288.016,E2 -11288.016} C_VEL
LIN {X 0,Y 399.357,Z 457.634,A -85,B 0,C 180,E1 -11289.965,E2 -11289.965} C_VEL
LIN {X 0,Y 398.489,Z 452.352,A -85,B 0,C 180,E1 -11292.914,E2 -11292.914} C_VEL
LIN {X 0,Y 397.677,Z 447.555,A -85,B 0,C 180,E1 -11295.728,E2 -11295.728} C_VEL
LIN {X 0,Y 397.15,Z 444.638,A -85,B 0,C 180,E1 -11297.572,E2 -11297.572} C_VEL
LIN {X 0,Y 397.128,Z 444.644,A -85,B 0,C 180,E1 -11301.138,E2 -11301.138} C_VEL
LIN {X 0,Y 397.115,Z 444.643,A -85,B 0,C 180,E1 -11304.496,E2 -11304.496} C_VEL
LIN {X 0,Y 397.107,Z 444.642,A -85,B 0,C 180,E1 -11307.931,E2 -11307.931} C_VEL
LIN {X 0,Y 397.122,Z 444.643,A -85,B 0,C 180,E1 -11311.456,E2 -11311.456} C_VEL
LIN {X 0,Y 397.147,Z 444.64,A -85,B 0,C 180,E1 -11314.487,E2 -11314.487} C_VEL
LIN {X 0,Y 397.103,Z 444.647,A -85,B 0,C 180,E1 -11317.085,E2 -11317.085} C_VEL
LIN {X 0,Y 397.142,Z 444.641,A -85,B 0,C 180,E1 -11320.353,E2 -11320.353} C_VEL
LIN {X 0,Y 397.16,Z 444.637,A -85,B 0,C 180,E1 -11323.553,E2 -11323.553} C_VEL
LIN {X 0,Y 397.222,Z 444.633,A -85,B 0,C 180,E1 -11326.703,E2 -11326.703} C_VEL
LIN {X 0,Y 397.213,Z 444.63,A -85,B 0,C 180,E1 -11329.809,E2 -11329.809} C_VEL
LIN {X 0,Y 397.358,Z 444.615,A -85,B 0,C 180,E1 -11332.888,E2 -11332.888} C_VEL
LIN {X 0,Y 397.251,Z 444.628,A -85,B 0,C 180,E1 -11334.925,E2 -11334.925} C_VEL
LIN {X 0,Y 397.446,Z 444.602,A -85,B 0,C 180,E1 -11337.973,E2 -11337.973} C_VEL
LIN {X 0,Y 397.574,Z 444.585,A -85,B 0,C 180,E1 -11340,E2 -11340} C_VEL
LIN {X 0,Y 397.378,Z 444.611,A -85,B 0,C 180,E1 -11343.042,E2 -11343.042} C_VEL
LIN {X 0,Y 397.355,Z 444.612,A -85,B 0,C 180,E1 -11346.592,E2 -11346.592} C_VEL
LIN {X 0,Y 397.247,Z 444.626,A -85,B 0,C 180,E1 -11349.162,E2 -11349.162} C_VEL
LIN {X 0,Y 397.213,Z 444.633,A -85,B 0,C 180,E1 -11352.259,E2 -11352.259} C_VEL
LIN {X 0,Y 397.173,Z 444.635,A -85,B 0,C 180,E1 -11355.393,E2 -11355.393} C_VEL
LIN {X 0,Y 397.157,Z 444.64,A -85,B 0,C 180,E1 -11358.574,E2 -11358.574} C_VEL
LIN {X 0,Y 397.092,Z 444.647,A -85,B 0,C 180,E1 -11361.819,E2 -11361.819} C_VEL
LIN {X 0,Y 397.152,Z 444.638,A -85,B 0,C 180,E1 -11365.132,E2 -11365.132} C_VEL
LIN {X 0,Y 397.157,Z 444.638,A -85,B 0,C 180,E1 -11367.777,E2 -11367.777} C_VEL
LIN {X 0,Y 397.074,Z 444.647,A -85,B 0,C 180,E1 -11370.883,E2 -11370.883} C_VEL
LIN {X 0,Y 397.123,Z 444.644,A -85,B 0,C 180,E1 -11374.494,E2 -11374.494} C_VEL
LIN {X 0,Y 397.102,Z 444.647,A -85,B 0,C 180,E1 -11378.275,E2 -11378.275} C_VEL
LIN {X 0,Y 397.087,Z 444.645,A -85,B 0,C 180,E1 -11380.909,E2 -11380.909} C_VEL
LIN {X 0,Y 397.102,Z 444.647,A -85,B 0,C 180,E1 -11383.649,E2 -11383.649} C_VEL
LIN {X 0,Y 397.103,Z 444.646,A -85,B 0,C 180,E1 -11386.521,E2 -11386.521} C_VEL
LIN {X 0,Y 397.12,Z 444.643,A -85,B 0,C 180,E1 -11389.552,E2 -11389.552} C_VEL
LIN {X 0,Y 397.099,Z 444.644,A -85,B 0,C 180,E1 -11392.791,E2 -11392.791} C_VEL
LIN {X 0,Y 397.119,Z 444.644,A -85,B 0,C 180,E1 -11396.283,E2 -11396.283} C_VEL
LIN {X 0,Y 397.115,Z 444.645,A -85,B 0,C 180,E1 -11400.134,E2 -11400.134} C_VEL
LIN {X 0,Y 397.196,Z 444.632,A -85,B 0,C 180,E1 -11402.611,E2 -11402.611} C_VEL
LIN {X 0,Y 397.135,Z 444.643,A -85,B 0,C 180,E1 -11405.982,E2 -11405.982} C_VEL
LIN {X 0,Y 397.141,Z 444.642,A -85,B 0,C 180,E1 -11409.705,E2 -11409.705} C_VEL
LIN {X 0,Y 397.185,Z 444.633,A -85,B 0,C 180,E1 -11412.845,E2 -11412.845} C_VEL
LIN {X 0,Y 397.232,Z 444.627,A -85,B 0,C 180,E1 -11416.703,E2 -11416.703} C_VEL
LIN {X 0,Y 397.221,Z 444.633,A -85,B 0,C 180,E1 -11419.809,E2 -11419.809} C_VEL
LIN {X 0,Y 397.321,Z 444.618,A -85,B 0,C 180,E1 -11422.888,E2 -11422.888} C_VEL
LIN {X 0,Y 397.251,Z 444.627,A -85,B 0,C 180,E1 -11424.925,E2 -11424.925} C_VEL
LIN {X 0,Y 397.455,Z 444.602,A -85,B 0,C 180,E1 -11427.973,E2 -11427.973} C_VEL
LIN {X 0,Y 397.583,Z 444.584,A -85,B 0,C 180,E1 -11430,E2 -11430} C_VEL
LIN {X 0,Y 397.379,Z 444.612,A -85,B 0,C 180,E1 -11433.041,E2 -11433.041} C_VEL
LIN {X 0,Y 397.373,Z 444.611,A -85,B 0,C 180,E1 -11436.091,E2 -11436.091} C_VEL
LIN {X 0,Y 397.255,Z 444.628,A -85,B 0,C 180,E1 -11439.162,E2 -11439.162} C_VEL
LIN {X 0,Y 397.223,Z 444.629,A -85,B 0,C 180,E1 -11442.258,E2 -11442.258} C_VEL
LIN {X 0,Y 397.182,Z 444.637,A -85,B 0,C 180,E1 -11445.392,E2 -11445.392} C_VEL
LIN {X 0,Y 397.165,Z 444.636,A -85,B 0,C 180,E1 -11448.573,E2 -11448.573} C_VEL
LIN {X 0,Y 397.094,Z 444.645,A -85,B 0,C 180,E1 -11451.919,E2 -11451.919} C_VEL
LIN {X 0,Y 397.155,Z 444.639,A -85,B 0,C 180,E1 -11455.512,E2 -11455.512} C_VEL
LIN {X 0,Y 397.136,Z 444.639,A -85,B 0,C 180,E1 -11456.331,E2 -11456.331} C_VEL
LIN {X 0,Y 396.467,Z 444.727,A -85,B 0,C 180,E1 -11457.178,E2 -11457.178} C_VEL
LIN {X 0,Y 393.592,Z 445.083,A -85,B 0,C 180,E1 -11458.553,E2 -11458.553} C_VEL
LIN {X 0,Y 391.152,Z 445.386,A -85,B 0,C 180,E1 -11459.665,E2 -11459.665} C_VEL
LIN {X 0,Y 390.099,Z 445.518,A -85,B 0,C 180,E1 -11460.524,E2 -11460.524} C_VEL
LIN {X 0,Y 390.011,Z 445.525,A -85,B 0,C 180,E1 -11460.816,E2 -11460.816} C_VEL
LIN {X 0,Y 390.019,Z 445.526,A -85,B 0,C 180,E1 -11464.013,E2 -11464.013} C_VEL
LIN {X 0,Y 389.799,Z 445.557,A -85,B 0,C 180,E1 -11466.511,E2 -11466.511} C_VEL
LIN {X 0,Y 389.461,Z 445.6,A -85,B 0,C 180,E1 -11469.167,E2 -11469.167} C_VEL
LIN {X 0,Y 389.274,Z 445.625,A -85,B 0,C 180,E1 -11470.687,E2 -11470.687} C_VEL
LIN {X 0,Y 389.18,Z 447.596,A -85,B 0,C 180,E1 -11473.331,E2 -11473.331} C_VEL
LIN {X 0,Y 389.085,Z 450.519,A -85,B 0,C 180,E1 -11476.655,E2 -11476.655} C_VEL
LIN {X 0,Y 389.016,Z 453.558,A -85,B 0,C 180,E1 -11480.03,E2 -11480.03} C_VEL
LIN {X 0,Y 393.139,Z 468.034,A -85,B 0,C 180,E1 -11480.744,E2 -11480.744} C_VEL
LIN {X 0,Y 396.803,Z 482.506,A -85,B 0,C 180,E1 -11481.643,E2 -11481.643} C_VEL
LIN {X 0,Y 396.189,Z 494.939,A -85,B 0,C 180,E1 -11482.426,E2 -11482.426} C_VEL
LIN {X 0,Y 395.186,Z 508.073,A -85,B 0,C 180,E1 -11483.459,E2 -11483.459} C_VEL
LIN {X 0,Y 394.027,Z 520.971,A -85,B 0,C 180,E1 -11484.728,E2 -11484.728} C_VEL
LIN {X 0,Y 392.898,Z 532.852,A -85,B 0,C 180,E1 -11486.168,E2 -11486.168} C_VEL
LIN {X 0,Y 391.916,Z 543.571,A -85,B 0,C 180,E1 -11487.758,E2 -11487.758} C_VEL
LIN {X 0,Y 390.852,Z 553.153,A -85,B 0,C 180,E1 -11489.501,E2 -11489.501} C_VEL
LIN {X 0,Y 390.217,Z 560.862,A -85,B 0,C 180,E1 -11491.227,E2 -11491.227} C_VEL
LIN {X 0,Y 389.637,Z 567.917,A -85,B 0,C 180,E1 -11493.196,E2 -11493.196} C_VEL
LIN {X 0,Y 389.258,Z 572.922,A -85,B 0,C 180,E1 -11494.974,E2 -11494.974} C_VEL
LIN {X 0,Y 388.995,Z 576.449,A -85,B 0,C 180,E1 -11496.579,E2 -11496.579} C_VEL
LIN {X 0,Y 388.83,Z 578.342,A -85,B 0,C 180,E1 -11497.693,E2 -11497.693} C_VEL
LIN {X 0,Y 388.704,Z 580.913,A -85,B 0,C 180,E1 -11499.908,E2 -11499.908} C_VEL
LIN {X 0,Y 388.667,Z 581.944,A -85,B 0,C 180,E1 -11502.097,E2 -11502.097} C_VEL
LIN {X 0,Y 388.743,Z 581.482,A -85,B 0,C 180,E1 -11504.265,E2 -11504.265} C_VEL
LIN {X 0,Y 388.906,Z 579.534,A -85,B 0,C 180,E1 -11506.412,E2 -11506.412} C_VEL
LIN {X 0,Y 389.108,Z 578.006,A -85,B 0,C 180,E1 -11507.482,E2 -11507.482} C_VEL
LIN {X 0,Y 389.529,Z 573.858,A -85,B 0,C 180,E1 -11509.605,E2 -11509.605} C_VEL
LIN {X 0,Y 390.106,Z 568.152,A -85,B 0,C 180,E1 -11511.713,E2 -11511.713} C_VEL
LIN {X 0,Y 390.865,Z 561.695,A -85,B 0,C 180,E1 -11513.547,E2 -11513.547} C_VEL
LIN {X 0,Y 391.856,Z 553.663,A -85,B 0,C 180,E1 -11515.371,E2 -11515.371} C_VEL
LIN {X 0,Y 392.792,Z 545.338,A -85,B 0,C 180,E1 -11516.923,E2 -11516.923} C_VEL
LIN {X 0,Y 394.129,Z 534.811,A -85,B 0,C 180,E1 -11518.53,E2 -11518.53} C_VEL
LIN {X 0,Y 395.355,Z 524.202,A -85,B 0,C 180,E1 -11519.872,E2 -11519.872} C_VEL
LIN {X 0,Y 396.661,Z 511.978,A -85,B 0,C 180,E1 -11521.142,E2 -11521.142} C_VEL
LIN {X 0,Y 397.844,Z 500.089,A -85,B 0,C 180,E1 -11522.142,E2 -11522.142} C_VEL
LIN {X 0,Y 398.959,Z 486.921,A -85,B 0,C 180,E1 -11523.029,E2 -11523.029} C_VEL
LIN {X 0,Y 398.57,Z 483.939,A -85,B 0,C 180,E1 -11523.241,E2 -11523.241} C_VEL
LIN {X 0,Y 394.648,Z 470.738,A -85,B 0,C 180,E1 -11524.253,E2 -11524.253} C_VEL
LIN {X 0,Y 389.97,Z 458.042,A -85,B 0,C 180,E1 -11525.137,E2 -11525.137} C_VEL
LIN {X 0,Y 389.892,Z 457.611,A -85,B 0,C 180,E1 -11525.171,E2 -11525.171} C_VEL
LIN {X 0,Y 389.945,Z 455.561,A -85,B 0,C 180,E1 -11528.29,E2 -11528.29} C_VEL
LIN {X 0,Y 390.061,Z 453.634,A -85,B 0,C 180,E1 -11531.431,E2 -11531.431} C_VEL
LIN {X 0,Y 390.206,Z 451.852,A -85,B 0,C 180,E1 -11534.605,E2 -11534.605} C_VEL
LIN {X 0,Y 390.416,Z 450.258,A -85,B 0,C 180,E1 -11537.82,E2 -11537.82} C_VEL
LIN {X 0,Y 390.481,Z 448.897,A -85,B 0,C 180,E1 -11541.098,E2 -11541.098} C_VEL
LIN {X 0,Y 390.434,Z 447.888,A -85,B 0,C 180,E1 -11544.457,E2 -11544.457} C_VEL
LIN {X 0,Y 390.405,Z 447.304,A -85,B 0,C 180,E1 -11548.106,E2 -11548.106} C_VEL
LIN {X 0,Y 390.365,Z 447.344,A -85,B 0,C 180,E1 -11551.474,E2 -11551.474} C_VEL
LIN {X 0,Y 390.466,Z 447.807,A -85,B 0,C 180,E1 -11554.112,E2 -11554.112} C_VEL
LIN {X 0,Y 390.697,Z 449.164,A -85,B 0,C 180,E1 -11557.706,E2 -11557.706} C_VEL
LIN {X 0,Y 390.989,Z 450.695,A -85,B 0,C 180,E1 -11560.323,E2 -11560.323} C_VEL
LIN {X 0,Y 391.357,Z 452.795,A -85,B 0,C 180,E1 -11563.032,E2 -11563.032} C_VEL
LIN {X 0,Y 391.834,Z 455.538,A -85,B 0,C 180,E1 -11565.844,E2 -11565.844} C_VEL
LIN {X 0,Y 392.391,Z 459.008,A -85,B 0,C 180,E1 -11568.786,E2 -11568.786} C_VEL
LIN {X 0,Y 392.512,Z 462.359,A -85,B 0,C 180,E1 -11571.195,E2 -11571.195} C_VEL
LIN {X 0,Y 392.229,Z 465.368,A -85,B 0,C 180,E1 -11573.113,E2 -11573.113} C_VEL
LIN {X 0,Y 391.49,Z 470.661,A -85,B 0,C 180,E1 -11576.186,E2 -11576.186} C_VEL
LIN {X 0,Y 390.806,Z 477.375,A -85,B 0,C 180,E1 -11579.767,E2 -11579.767} C_VEL
LIN {X 0,Y 390.196,Z 484.39,A -85,B 0,C 180,E1 -11583.238,E2 -11583.238} C_VEL
LIN {X 0,Y 389.672,Z 491.941,A -85,B 0,C 180,E1 -11586.768,E2 -11586.768} C_VEL
LIN {X 0,Y 393.444,Z 507.36,A -85,B 0,C 180,E1 -11587.616,E2 -11587.616} C_VEL
LIN {X 0,Y 395.776,Z 521.391,A -85,B 0,C 180,E1 -11588.481,E2 -11588.481} C_VEL
LIN {X 0,Y 396.956,Z 534.52,A -85,B 0,C 180,E1 -11589.398,E2 -11589.398} C_VEL
LIN {X 0,Y 395.656,Z 547.923,A -85,B 0,C 180,E1 -11590.397,E2 -11590.397} C_VEL
LIN {X 0,Y 394.385,Z 560.48,A -85,B 0,C 180,E1 -11591.561,E2 -11591.561} C_VEL
LIN {X 0,Y 392.945,Z 573.001,A -85,B 0,C 180,E1 -11592.97,E2 -11592.97} C_VEL
LIN {X 0,Y 391.793,Z 583.37,A -85,B 0,C 180,E1 -11594.391,E2 -11594.391} C_VEL
LIN {X 0,Y 390.835,Z 592.842,A -85,B 0,C 180,E1 -11595.951,E2 -11595.951} C_VEL
LIN {X 0,Y 390.073,Z 600.788,A -85,B 0,C 180,E1 -11597.514,E2 -11597.514} C_VEL
LIN {X 0,Y 389.507,Z 607.426,A -85,B 0,C 180,E1 -11599.079,E2 -11599.079} C_VEL
LIN {X 0,Y 389.132,Z 612.964,A -85,B 0,C 180,E1 -11600.645,E2 -11600.645} C_VEL
LIN {X 0,Y 388.908,Z 618.854,A -85,B 0,C 180,E1 -11602.733,E2 -11602.733} C_VEL
LIN {X 0,Y 388.78,Z 623.132,A -85,B 0,C 180,E1 -11604.814,E2 -11604.814} C_VEL
LIN {X 0,Y 388.751,Z 625.901,A -85,B 0,C 180,E1 -11606.891,E2 -11606.891} C_VEL
LIN {X 0,Y 388.84,Z 626.754,A -85,B 0,C 180,E1 -11607.928,E2 -11607.928} C_VEL
LIN {X 0,Y 388.797,Z 627.4,A -85,B 0,C 180,E1 -11610,E2 -11610} C_VEL
LIN {X 0,Y 388.841,Z 626.65,A -85,B 0,C 180,E1 -11612.072,E2 -11612.072} C_VEL
LIN {X 0,Y 388.722,Z 624.473,A -85,B 0,C 180,E1 -11614.147,E2 -11614.147} C_VEL
LIN {X 0,Y 388.833,Z 620.838,A -85,B 0,C 180,E1 -11616.226,E2 -11616.226} C_VEL
LIN {X 0,Y 388.907,Z 617.071,A -85,B 0,C 180,E1 -11617.789,E2 -11617.789} C_VEL
LIN {X 0,Y 389.131,Z 612.375,A -85,B 0,C 180,E1 -11619.355,E2 -11619.355} C_VEL
LIN {X 0,Y 389.613,Z 605.519,A -85,B 0,C 180,E1 -11621.181,E2 -11621.181} C_VEL
LIN {X 0,Y 390.33,Z 596.985,A -85,B 0,C 180,E1 -11623.007,E2 -11623.007} C_VEL
LIN {X 0,Y 391.018,Z 588.075,A -85,B 0,C 180,E1 -11624.574,E2 -11624.574} C_VEL
LIN {X 0,Y 392.064,Z 577.329,A -85,B 0,C 180,E1 -11626.131,E2 -11626.131} C_VEL
LIN {X 0,Y 393.241,Z 565.352,A -85,B 0,C 180,E1 -11627.553,E2 -11627.553} C_VEL
LIN {X 0,Y 394.393,Z 553.381,A -85,B 0,C 180,E1 -11628.708,E2 -11628.708} C_VEL
LIN {X 0,Y 395.51,Z 540.162,A -85,B 0,C 180,E1 -11629.732,E2 -11629.732} C_VEL
LIN {X 0,Y 396.006,Z 534.32,A -85,B 0,C 180,E1 -11630.111,E2 -11630.111} C_VEL
LIN {X 0,Y 394.044,Z 520.023,A -85,B 0,C 180,E1 -11631,E2 -11631} C_VEL
LIN {X 0,Y 391.411,Z 504.764,A -85,B 0,C 180,E1 -11631.748,E2 -11631.748} C_VEL
LIN {X 0,Y 389.648,Z 495.634,A -85,B 0,C 180,E1 -11632.123,E2 -11632.123} C_VEL
LIN {X 0,Y 390.133,Z 487.714,A -85,B 0,C 180,E1 -11635.747,E2 -11635.747} C_VEL
LIN {X 0,Y 390.658,Z 480.619,A -85,B 0,C 180,E1 -11639.06,E2 -11639.06} C_VEL
LIN {X 0,Y 391.359,Z 473.27,A -85,B 0,C 180,E1 -11642.597,E2 -11642.597} C_VEL
LIN {X 0,Y 392.001,Z 465.884,A -85,B 0,C 180,E1 -11646.273,E2 -11646.273} C_VEL
LIN {X 0,Y 392.459,Z 460.969,A -85,B 0,C 180,E1 -11648.811,E2 -11648.811} C_VEL
LIN {X 0,Y 392.081,Z 456.663,A -85,B 0,C 180,E1 -11651.163,E2 -11651.163} C_VEL
LIN {X 0,Y 391.057,Z 450.945,A -85,B 0,C 180,E1 -11654.498,E2 -11654.498} C_VEL
LIN {X 0,Y 390.112,Z 445.514,A -85,B 0,C 180,E1 -11657.899,E2 -11657.899} C_VEL
LIN {X 0,Y 390.087,Z 445.522,A -85,B 0,C 180,E1 -11660.907,E2 -11660.907} C_VEL
LIN {X 0,Y 390.08,Z 445.521,A -85,B 0,C 180,E1 -11664.793,E2 -11664.793} C_VEL
LIN {X 0,Y 390.044,Z 445.524,A -85,B 0,C 180,E1 -11668.498,E2 -11668.498} C_VEL
LIN {X 0,Y 390.112,Z 445.514,A -85,B 0,C 180,E1 -11672.07,E2 -11672.07} C_VEL
LIN {X 0,Y 390.074,Z 445.52,A -85,B 0,C 180,E1 -11675.519,E2 -11675.519} C_VEL
LIN {X 0,Y 390.05,Z 445.526,A -85,B 0,C 180,E1 -11678.878,E2 -11678.878} C_VEL
LIN {X 0,Y 390.122,Z 445.513,A -85,B 0,C 180,E1 -11682.167,E2 -11682.167} C_VEL
LIN {X 0,Y 390.137,Z 445.512,A -85,B 0,C 180,E1 -11685.393,E2 -11685.393} C_VEL
LIN {X 0,Y 390.143,Z 445.514,A -85,B 0,C 180,E1 -11688.571,E2 -11688.571} C_VEL
LIN {X 0,Y 390.338,Z 445.487,A -85,B 0,C 180,E1 -11691.993,E2 -11691.993} C_VEL
LIN {X 0,Y 390.222,Z 445.504,A -85,B 0,C 180,E1 -11694.834,E2 -11694.834} C_VEL
LIN {X 0,Y 390.415,Z 445.478,A -85,B 0,C 180,E1 -11697.937,E2 -11697.937} C_VEL
LIN {X 0,Y 390.544,Z 445.461,A -85,B 0,C 180,E1 -11700,E2 -11700} C_VEL
LIN {X 0,Y 390.312,Z 445.491,A -85,B 0,C 180,E1 -11703.097,E2 -11703.097} C_VEL
LIN {X 0,Y 390.312,Z 445.49,A -85,B 0,C 180,E1 -11706.586,E2 -11706.586} C_VEL
LIN {X 0,Y 390.199,Z 445.503,A -85,B 0,C 180,E1 -11709.329,E2 -11709.329} C_VEL
LIN {X 0,Y 390.189,Z 445.504,A -85,B 0,C 180,E1 -11713.439,E2 -11713.439} C_VEL
LIN {X 0,Y 390.143,Z 445.51,A -85,B 0,C 180,E1 -11717.308,E2 -11717.308} C_VEL
LIN {X 0,Y 390.082,Z 445.522,A -85,B 0,C 180,E1 -11720.471,E2 -11720.471} C_VEL
LIN {X 0,Y 390.085,Z 445.518,A -85,B 0,C 180,E1 -11723.351,E2 -11723.351} C_VEL
LIN {X 0,Y 390.109,Z 445.516,A -85,B 0,C 180,E1 -11726.769,E2 -11726.769} C_VEL
LIN {X 0,Y 390.035,Z 445.528,A -85,B 0,C 180,E1 -11730.3,E2 -11730.3} C_VEL
LIN {X 0,Y 390.065,Z 445.524,A -85,B 0,C 180,E1 -11734.025,E2 -11734.025} C_VEL
LIN {X 0,Y 390.042,Z 445.524,A -85,B 0,C 180,E1 -11737.552,E2 -11737.552} C_VEL
LIN {X 0,Y 390.054,Z 445.521,A -85,B 0,C 180,E1 -11740.822,E2 -11740.822} C_VEL
LIN {X 0,Y 390.055,Z 445.525,A -85,B 0,C 180,E1 -11743.887,E2 -11743.887} C_VEL
LIN {X 0,Y 390.079,Z 445.522,A -85,B 0,C 180,E1 -11747.621,E2 -11747.621} C_VEL
LIN {X 0,Y 390.095,Z 445.517,A -85,B 0,C 180,E1 -11750.909,E2 -11750.909} C_VEL
LIN {X 0,Y 390.086,Z 445.517,A -85,B 0,C 180,E1 -11754.794,E2 -11754.794} C_VEL
LIN {X 0,Y 390.035,Z 445.528,A -85,B 0,C 180,E1 -11757.876,E2 -11757.876} C_VEL
LIN {X 0,Y 390.067,Z 445.52,A -85,B 0,C 180,E1 -11760.892,E2 -11760.892} C_VEL
LIN {X 0,Y 390.113,Z 445.515,A -85,B 0,C 180,E1 -11764.383,E2 -11764.383} C_VEL
LIN {X 0,Y 390.043,Z 445.527,A -85,B 0,C 180,E1 -11767.766,E2 -11767.766} C_VEL
LIN {X 0,Y 390.108,Z 445.516,A -85,B 0,C 180,E1 -11771.078,E2 -11771.078} C_VEL
LIN {X 0,Y 390.143,Z 445.511,A -85,B 0,C 180,E1 -11774.324,E2 -11774.324} C_VEL
LIN {X 0,Y 390.174,Z 445.511,A -85,B 0,C 180,E1 -11777.517,E2 -11777.517} C_VEL
LIN {X 0,Y 390.207,Z 445.502,A -85,B 0,C 180,E1 -11780.671,E2 -11780.671} C_VEL
LIN {X 0,Y 390.303,Z 445.494,A -85,B 0,C 180,E1 -11783.798,E2 -11783.798} C_VEL
LIN {X 0,Y 390.424,Z 445.477,A -85,B 0,C 180,E1 -11787.937,E2 -11787.937} C_VEL
LIN {X 0,Y 390.552,Z 445.46,A -85,B 0,C 180,E1 -11790,E2 -11790} C_VEL
LIN {X 0,Y 390.314,Z 445.493,A -85,B 0,C 180,E1 -11793.096,E2 -11793.096} C_VEL
LIN {X 0,Y 390.326,Z 445.488,A -85,B 0,C 180,E1 -11796.202,E2 -11796.202} C_VEL
LIN {X 0,Y 390.207,Z 445.507,A -85,B 0,C 180,E1 -11799.329,E2 -11799.329} C_VEL
LIN {X 0,Y 390.174,Z 445.507,A -85,B 0,C 180,E1 -11802.483,E2 -11802.483} C_VEL
LIN {X 0,Y 390.142,Z 445.513,A -85,B 0,C 180,E1 -11805.676,E2 -11805.676} C_VEL
LIN {X 0,Y 390.108,Z 445.518,A -85,B 0,C 180,E1 -11808.922,E2 -11808.922} C_VEL
LIN {X 0,Y 390.042,Z 445.523,A -85,B 0,C 180,E1 -11812.234,E2 -11812.234} C_VEL
LIN {X 0,Y 390.121,Z 445.514,A -85,B 0,C 180,E1 -11815.743,E2 -11815.743} C_VEL
LIN {X 0,Y 390.06,Z 445.524,A -85,B 0,C 180,E1 -11819.109,E2 -11819.109} C_VEL
LIN {X 0,Y 390.011,Z 445.525,A -85,B 0,C 180,E1 -11820.816,E2 -11820.816} C_VEL
LIN {X 0,Y 389.334,Z 445.612,A -85,B 0,C 180,E1 -11821.678,E2 -11821.678} C_VEL
LIN {X 0,Y 386.463,Z 445.972,A -85,B 0,C 180,E1 -11823.078,E2 -11823.078} C_VEL
LIN {X 0,Y 384.023,Z 446.275,A -85,B 0,C 180,E1 -11824.21,E2 -11824.21} C_VEL
LIN {X 0,Y 382.957,Z 446.41,A -85,B 0,C 180,E1 -11825.086,E2 -11825.086} C_VEL
LIN {X 0,Y 382.86,Z 446.417,A -85,B 0,C 180,E1 -11825.383,E2 -11825.383} C_VEL
LIN {X 0,Y 382.46,Z 446.472,A -85,B 0,C 180,E1 -11828.665,E2 -11828.665} C_VEL
LIN {X 0,Y 382.137,Z 446.731,A -85,B 0,C 180,E1 -11831.458,E2 -11831.458} C_VEL
LIN {X 0,Y 382.079,Z 449.192,A -85,B 0,C 180,E1 -11834.344,E2 -11834.344} C_VEL
LIN {X 0,Y 381.992,Z 451.872,A -85,B 0,C 180,E1 -11837.385,E2 -11837.385} C_VEL
LIN {X 0,Y 381.962,Z 453.911,A -85,B 0,C 180,E1 -11839.666,E2 -11839.666} C_VEL
LIN {X 0,Y 386.16,Z 468.747,A -85,B 0,C 180,E1 -11840.418,E2 -11840.418} C_VEL
LIN {X 0,Y 389.648,Z 482.375,A -85,B 0,C 180,E1 -11841.289,E2 -11841.289} C_VEL
LIN {X 0,Y 390.084,Z 485.553,A -85,B 0,C 180,E1 -11841.503,E2 -11841.503} C_VEL
LIN {X 0,Y 389.095,Z 499.033,A -85,B 0,C 180,E1 -11842.41,E2 -11842.41} C_VEL
LIN {X 0,Y 388.083,Z 511.437,A -85,B 0,C 180,E1 -11843.462,E2 -11843.462} C_VEL
LIN {X 0,Y 386.936,Z 523.454,A -85,B 0,C 180,E1 -11844.712,E2 -11844.712} C_VEL
LIN {X 0,Y 385.888,Z 534.396,A -85,B 0,C 180,E1 -11846.099,E2 -11846.099} C_VEL
LIN {X 0,Y 384.872,Z 544.909,A -85,B 0,C 180,E1 -11847.723,E2 -11847.723} C_VEL
LIN {X 0,Y 383.842,Z 553.75,A -85,B 0,C 180,E1 -11849.377,E2 -11849.377} C_VEL
LIN {X 0,Y 383.142,Z 561.749,A -85,B 0,C 180,E1 -11851.216,E2 -11851.216} C_VEL
LIN {X 0,Y 382.541,Z 568.81,A -85,B 0,C 180,E1 -11853.249,E2 -11853.249} C_VEL
LIN {X 0,Y 382.172,Z 573.516,A -85,B 0,C 180,E1 -11854.978,E2 -11854.978} C_VEL
LIN {X 0,Y 381.863,Z 577.604,A -85,B 0,C 180,E1 -11856.957,E2 -11856.957} C_VEL
LIN {X 0,Y 381.67,Z 579.787,A -85,B 0,C 180,E1 -11858.39,E2 -11858.39} C_VEL
LIN {X 0,Y 381.621,Z 581.834,A -85,B 0,C 180,E1 -11860.64,E2 -11860.64} C_VEL
LIN {X 0,Y 381.586,Z 582.368,A -85,B 0,C 180,E1 -11862.861,E2 -11862.861} C_VEL
LIN {X 0,Y 381.694,Z 581.439,A -85,B 0,C 180,E1 -11865.062,E2 -11865.062} C_VEL
LIN {X 0,Y 381.992,Z 579.071,A -85,B 0,C 180,E1 -11867.245,E2 -11867.245} C_VEL
LIN {X 0,Y 382.431,Z 575.204,A -85,B 0,C 180,E1 -11869.41,E2 -11869.41} C_VEL
LIN {X 0,Y 383.023,Z 569.761,A -85,B 0,C 180,E1 -11871.559,E2 -11871.559} C_VEL
LIN {X 0,Y 383.67,Z 564.571,A -85,B 0,C 180,E1 -11873.162,E2 -11873.162} C_VEL
LIN {X 0,Y 384.608,Z 557.114,A -85,B 0,C 180,E1 -11875.02,E2 -11875.02} C_VEL
LIN {X 0,Y 385.618,Z 549.396,A -85,B 0,C 180,E1 -11876.604,E2 -11876.604} C_VEL
LIN {X 0,Y 386.902,Z 539.42,A -85,B 0,C 180,E1 -11878.289,E2 -11878.289} C_VEL
LIN {X 0,Y 388.249,Z 528.941,A -85,B 0,C 180,E1 -11879.741,E2 -11879.741} C_VEL
LIN {X 0,Y 389.564,Z 517.647,A -85,B 0,C 180,E1 -11881.034,E2 -11881.034} C_VEL
LIN {X 0,Y 390.885,Z 505.317,A -85,B 0,C 180,E1 -11882.189,E2 -11882.189} C_VEL
LIN {X 0,Y 392.157,Z 492.284,A -85,B 0,C 180,E1 -11883.165,E2 -11883.165} C_VEL
LIN {X 0,Y 392.463,Z 487.134,A -85,B 0,C 180,E1 -11883.503,E2 -11883.503} C_VEL
LIN {X 0,Y 388.89,Z 474.459,A -85,B 0,C 180,E1 -11884.535,E2 -11884.535} C_VEL
LIN {X 0,Y 384.061,Z 461.452,A -85,B 0,C 180,E1 -11885.529,E2 -11885.529} C_VEL
LIN {X 0,Y 382.921,Z 458.698,A -85,B 0,C 180,E1 -11885.727,E2 -11885.727} C_VEL
LIN {X 0,Y 382.857,Z 458.202,A -85,B 0,C 180,E1 -11885.794,E2 -11885.794} C_VEL
LIN {X 0,Y 382.931,Z 456.515,A -85,B 0,C 180,E1 -11888.443,E2 -11888.443} C_VEL
LIN {X 0,Y 383.048,Z 454.612,A -85,B 0,C 180,E1 -11891.643,E2 -11891.643} C_VEL
LIN {X 0,Y 383.207,Z 452.877,A -85,B 0,C 180,E1 -11894.878,E2 -11894.878} C_VEL
LIN {X 0,Y 383.442,Z 451.338,A -85,B 0,C 180,E1 -11898.155,E2 -11898.155} C_VEL
LIN {X 0,Y 383.485,Z 450.073,A -85,B 0,C 180,E1 -11901.502,E2 -11901.502} C_VEL
LIN {X 0,Y 383.467,Z 449.158,A -85,B 0,C 180,E1 -11904.931,E2 -11904.931} C_VEL
LIN {X 0,Y 383.433,Z 448.721,A -85,B 0,C 180,E1 -11908.461,E2 -11908.461} C_VEL
LIN {X 0,Y 383.451,Z 448.917,A -85,B 0,C 180,E1 -11912.108,E2 -11912.108} C_VEL
LIN {X 0,Y 383.538,Z 449.477,A -85,B 0,C 180,E1 -11914.614,E2 -11914.614} C_VEL
LIN {X 0,Y 383.798,Z 450.885,A -85,B 0,C 180,E1 -11918.058,E2 -11918.058} C_VEL
LIN {X 0,Y 384.212,Z 453.001,A -85,B 0,C 180,E1 -11921.413,E2 -11921.413} C_VEL
LIN {X 0,Y 384.672,Z 455.721,A -85,B 0,C 180,E1 -11924.56,E2 -11924.56} C_VEL
LIN {X 0,Y 385.202,Z 458.906,A -85,B 0,C 180,E1 -11927.542,E2 -11927.542} C_VEL
LIN {X 0,Y 385.584,Z 462.5,A -85,B 0,C 180,E1 -11930.362,E2 -11930.362} C_VEL
LIN {X 0,Y 385.394,Z 465.435,A -85,B 0,C 180,E1 -11932.346,E2 -11932.346} C_VEL
LIN {X 0,Y 384.489,Z 471.694,A -85,B 0,C 180,E1 -11936.117,E2 -11936.117} C_VEL
LIN {X 0,Y 383.85,Z 477.644,A -85,B 0,C 180,E1 -11939.377,E2 -11939.377} C_VEL
LIN {X 0,Y 383.129,Z 485.357,A -85,B 0,C 180,E1 -11943.294,E2 -11943.294} C_VEL
LIN {X 0,Y 382.669,Z 491.344,A -85,B 0,C 180,E1 -11946.169,E2 -11946.169} C_VEL
LIN {X 0,Y 386.671,Z 507.153,A -85,B 0,C 180,E1 -11947.104,E2 -11947.104} C_VEL
LIN {X 0,Y 389.066,Z 521.12,A -85,B 0,C 180,E1 -11948.012,E2 -11948.012} C_VEL
LIN {X 0,Y 390.268,Z 535.048,A -85,B 0,C 180,E1 -11949.029,E2 -11949.029} C_VEL
LIN {X 0,Y 389.283,Z 545.88,A -85,B 0,C 180,E1 -11949.85,E2 -11949.85} C_VEL
LIN {X 0,Y 387.964,Z 558.113,A -85,B 0,C 180,E1 -11950.97,E2 -11950.97} C_VEL
LIN {X 0,Y 386.368,Z 570.896,A -85,B 0,C 180,E1 -11952.398,E2 -11952.398} C_VEL
LIN {X 0,Y 385.098,Z 581.479,A -85,B 0,C 180,E1 -11953.841,E2 -11953.841} C_VEL
LIN {X 0,Y 384.004,Z 591.327,A -85,B 0,C 180,E1 -11955.452,E2 -11955.452} C_VEL
LIN {X 0,Y 383.101,Z 600.55,A -85,B 0,C 180,E1 -11957.283,E2 -11957.283} C_VEL
LIN {X 0,Y 382.487,Z 607.176,A -85,B 0,C 180,E1 -11958.876,E2 -11958.876} C_VEL
LIN {X 0,Y 382.076,Z 612.667,A -85,B 0,C 180,E1 -11960.471,E2 -11960.471} C_VEL
LIN {X 0,Y 381.823,Z 618.514,A -85,B 0,C 180,E1 -11962.597,E2 -11962.597} C_VEL
LIN {X 0,Y 381.684,Z 622.758,A -85,B 0,C 180,E1 -11964.718,E2 -11964.718} C_VEL
LIN {X 0,Y 381.654,Z 625.501,A -85,B 0,C 180,E1 -11966.833,E2 -11966.833} C_VEL
LIN {X 0,Y 381.771,Z 626.345,A -85,B 0,C 180,E1 -11967.89,E2 -11967.89} C_VEL
LIN {X 0,Y 381.724,Z 626.966,A -85,B 0,C 180,E1 -11970,E2 -11970} C_VEL
LIN {X 0,Y 381.772,Z 626.187,A -85,B 0,C 180,E1 -11972.11,E2 -11972.11} C_VEL
LIN {X 0,Y 381.648,Z 623.977,A -85,B 0,C 180,E1 -11974.224,E2 -11974.224} C_VEL
LIN {X 0,Y 381.764,Z 620.305,A -85,B 0,C 180,E1 -11976.341,E2 -11976.341} C_VEL
LIN {X 0,Y 381.913,Z 615.047,A -85,B 0,C 180,E1 -11978.466,E2 -11978.466} C_VEL
LIN {X 0,Y 382.179,Z 609.916,A -85,B 0,C 180,E1 -11980.061,E2 -11980.061} C_VEL
LIN {X 0,Y 382.782,Z 602.58,A -85,B 0,C 180,E1 -11981.92,E2 -11981.92} C_VEL
LIN {X 0,Y 383.301,Z 594.966,A -85,B 0,C 180,E1 -11983.499,E2 -11983.499} C_VEL
LIN {X 0,Y 384.239,Z 585.636,A -85,B 0,C 180,E1 -11985.108,E2 -11985.108} C_VEL
LIN {X 0,Y 385.308,Z 575.482,A -85,B 0,C 180,E1 -11986.559,E2 -11986.559} C_VEL
LIN {X 0,Y 386.444,Z 564.39,A -85,B 0,C 180,E1 -11987.872,E2 -11987.872} C_VEL
LIN {X 0,Y 387.676,Z 551.226,A -85,B 0,C 180,E1 -11989.136,E2 -11989.136} C_VEL
LIN {X 0,Y 388.797,Z 538.871,A -85,B 0,C 180,E1 -11990.087,E2 -11990.087} C_VEL
LIN {X 0,Y 388.984,Z 534.237,A -85,B 0,C 180,E1 -11990.404,E2 -11990.404} C_VEL
LIN {X 0,Y 387.126,Z 520.441,A -85,B 0,C 180,E1 -11991.289,E2 -11991.289} C_VEL
LIN {X 0,Y 384.523,Z 505.264,A -85,B 0,C 180,E1 -11992.064,E2 -11992.064} C_VEL
LIN {X 0,Y 382.607,Z 495.278,A -85,B 0,C 180,E1 -11992.491,E2 -11992.491} C_VEL
LIN {X 0,Y 383.141,Z 487.528,A -85,B 0,C 180,E1 -11996.118,E2 -11996.118} C_VEL
LIN {X 0,Y 383.727,Z 480.198,A -85,B 0,C 180,E1 -11999.637,E2 -11999.637} C_VEL
LIN {X 0,Y 384.413,Z 472.83,A -85,B 0,C 180,E1 -12003.262,E2 -12003.262} C_VEL
LIN {X 0,Y 385.022,Z 466.367,A -85,B 0,C 180,E1 -12006.568,E2 -12006.568} C_VEL
LIN {X 0,Y 385.435,Z 461.771,A -85,B 0,C 180,E1 -12008.98,E2 -12008.98} C_VEL
LIN {X 0,Y 385.122,Z 458.039,A -85,B 0,C 180,E1 -12011.067,E2 -12011.067} C_VEL
LIN {X 0,Y 384.095,Z 452.287,A -85,B 0,C 180,E1 -12014.471,E2 -12014.471} C_VEL
LIN {X 0,Y 383.072,Z 446.392,A -85,B 0,C 180,E1 -12018.225,E2 -12018.225} C_VEL
LIN {X 0,Y 383.001,Z 446.404,A -85,B 0,C 180,E1 -12021.399,E2 -12021.399} C_VEL
LIN {X 0,Y 383.02,Z 446.397,A -85,B 0,C 180,E1 -12024.044,E2 -12024.044} C_VEL
LIN {X 0,Y 383.033,Z 446.396,A -85,B 0,C 180,E1 -12027.853,E2 -12027.853} C_VEL
LIN {X 0,Y 383.059,Z 446.393,A -85,B 0,C 180,E1 -12031.72,E2 -12031.72} C_VEL
LIN {X 0,Y 383.047,Z 446.398,A -85,B 0,C 180,E1 -12035.04,E2 -12035.04} C_VEL
LIN {X 0,Y 382.987,Z 446.404,A -85,B 0,C 180,E1 -12038.469,E2 -12038.469} C_VEL
LIN {X 0,Y 383.057,Z 446.392,A -85,B 0,C 180,E1 -12041.826,E2 -12041.826} C_VEL
LIN {X 0,Y 383.104,Z 446.39,A -85,B 0,C 180,E1 -12045.118,E2 -12045.118} C_VEL
LIN {X 0,Y 383.092,Z 446.391,A -85,B 0,C 180,E1 -12048.358,E2 -12048.358} C_VEL
LIN {X 0,Y 383.298,Z 446.363,A -85,B 0,C 180,E1 -12051.933,E2 -12051.933} C_VEL
LIN {X 0,Y 383.194,Z 446.381,A -85,B 0,C 180,E1 -12054.739,E2 -12054.739} C_VEL
LIN {X 0,Y 383.382,Z 446.353,A -85,B 0,C 180,E1 -12057.899,E2 -12057.899} C_VEL
LIN {X 0,Y 383.513,Z 446.337,A -85,B 0,C 180,E1 -12060,E2 -12060} C_VEL
LIN {X 0,Y 383.248,Z 446.37,A -85,B 0,C 180,E1 -12063.154,E2 -12063.154} C_VEL
LIN {X 0,Y 383.273,Z 446.368,A -85,B 0,C 180,E1 -12066.578,E2 -12066.578} C_VEL
LIN {X 0,Y 383.254,Z 446.373,A -85,B 0,C 180,E1 -12068.436,E2 -12068.436} C_VEL
LIN {X 0,Y 383.091,Z 446.389,A -85,B 0,C 180,E1 -12071.643,E2 -12071.643} C_VEL
LIN {X 0,Y 383.104,Z 446.389,A -85,B 0,C 180,E1 -12074.882,E2 -12074.882} C_VEL
LIN {X 0,Y 383.084,Z 446.393,A -85,B 0,C 180,E1 -12078.173,E2 -12078.173} C_VEL
LIN {X 0,Y 382.988,Z 446.402,A -85,B 0,C 180,E1 -12081.532,E2 -12081.532} C_VEL
LIN {X 0,Y 383.048,Z 446.395,A -85,B 0,C 180,E1 -12084.961,E2 -12084.961} C_VEL
LIN {X 0,Y 383.036,Z 446.399,A -85,B 0,C 180,E1 -12088.493,E2 -12088.493} C_VEL
LIN {X 0,Y 383.006,Z 446.404,A -85,B 0,C 180,E1 -12092.15,E2 -12092.15} C_VEL
LIN {X 0,Y 383.015,Z 446.4,A -85,B 0,C 180,E1 -12094.669,E2 -12094.669} C_VEL
LIN {X 0,Y 382.998,Z 446.405,A -85,B 0,C 180,E1 -12097.905,E2 -12097.905} C_VEL
LIN {X 0,Y 382.982,Z 446.402,A -85,B 0,C 180,E1 -12101.348,E2 -12101.348} C_VEL
LIN {X 0,Y 382.996,Z 446.403,A -85,B 0,C 180,E1 -12104.304,E2 -12104.304} C_VEL
LIN {X 0,Y 383.038,Z 446.396,A -85,B 0,C 180,E1 -12107.245,E2 -12107.245} C_VEL
LIN {X 0,Y 383.021,Z 446.399,A -85,B 0,C 180,E1 -12110.413,E2 -12110.413} C_VEL
LIN {X 0,Y 383.027,Z 446.4,A -85,B 0,C 180,E1 -12114.045,E2 -12114.045} C_VEL
LIN {X 0,Y 382.989,Z 446.405,A -85,B 0,C 180,E1 -12117.578,E2 -12117.578} C_VEL
LIN {X 0,Y 382.999,Z 446.402,A -85,B 0,C 180,E1 -12120.301,E2 -12120.301} C_VEL
LIN {X 0,Y 383.058,Z 446.392,A -85,B 0,C 180,E1 -12122.699,E2 -12122.699} C_VEL
LIN {X 0,Y 383.036,Z 446.397,A -85,B 0,C 180,E1 -12126.193,E2 -12126.193} C_VEL
LIN {X 0,Y 383.058,Z 446.397,A -85,B 0,C 180,E1 -12129.599,E2 -12129.599} C_VEL
LIN {X 0,Y 383.108,Z 446.387,A -85,B 0,C 180,E1 -12132.932,E2 -12132.932} C_VEL
LIN {X 0,Y 383.128,Z 446.383,A -85,B 0,C 180,E1 -12136.464,E2 -12136.464} C_VEL
LIN {X 0,Y 383.154,Z 446.381,A -85,B 0,C 180,E1 -12140.498,E2 -12140.498} C_VEL
LIN {X 0,Y 383.259,Z 446.372,A -85,B 0,C 180,E1 -12143.683,E2 -12143.683} C_VEL
LIN {X 0,Y 383.392,Z 446.353,A -85,B 0,C 180,E1 -12147.899,E2 -12147.899} C_VEL
LIN {X 0,Y 383.522,Z 446.335,A -85,B 0,C 180,E1 -12150,E2 -12150} C_VEL
LIN {X 0,Y 383.251,Z 446.372,A -85,B 0,C 180,E1 -12153.154,E2 -12153.154} C_VEL
LIN {X 0,Y 383.282,Z 446.365,A -85,B 0,C 180,E1 -12156.316,E2 -12156.316} C_VEL
LIN {X 0,Y 383.154,Z 446.384,A -85,B 0,C 180,E1 -12159.502,E2 -12159.502} C_VEL
LIN {X 0,Y 383.128,Z 446.386,A -85,B 0,C 180,E1 -12163.536,E2 -12163.536} C_VEL
LIN {X 0,Y 383.098,Z 446.391,A -85,B 0,C 180,E1 -12167.454,E2 -12167.454} C_VEL
LIN {X 0,Y 383.031,Z 446.398,A -85,B 0,C 180,E1 -12170.647,E2 -12170.647} C_VEL
LIN {X 0,Y 383.036,Z 446.396,A -85,B 0,C 180,E1 -12173.807,E2 -12173.807} C_VEL
LIN {X 0,Y 383.082,Z 446.39,A -85,B 0,C 180,E1 -12176.123,E2 -12176.123} C_VEL
LIN {X 0,Y 382.993,Z 446.402,A -85,B 0,C 180,E1 -12179.699,E2 -12179.699} C_VEL
LIN {X 0,Y 382.978,Z 446.404,A -85,B 0,C 180,E1 -12182.419,E2 -12182.419} C_VEL
LIN {X 0,Y 382.86,Z 446.417,A -85,B 0,C 180,E1 -12185.383,E2 -12185.383} C_VEL
LIN {X 0,Y 382.137,Z 446.51,A -85,B 0,C 180,E1 -12186.259,E2 -12186.259} C_VEL
LIN {X 0,Y 379.139,Z 446.887,A -85,B 0,C 180,E1 -12187.679,E2 -12187.679} C_VEL
LIN {X 0,Y 376.565,Z 447.21,A -85,B 0,C 180,E1 -12188.826,E2 -12188.826} C_VEL
LIN {X 0,Y 375.39,Z 447.355,A -85,B 0,C 180,E1 -12189.716,E2 -12189.716} C_VEL
LIN {X 0,Y 375.256,Z 447.37,A -85,B 0,C 180,E1 -12190.019,E2 -12190.019} C_VEL
LIN {X 0,Y 375.088,Z 447.461,A -85,B 0,C 180,E1 -12191.454,E2 -12191.454} C_VEL
LIN {X 0,Y 375.021,Z 450.125,A -85,B 0,C 180,E1 -12194.591,E2 -12194.591} C_VEL
LIN {X 0,Y 374.919,Z 452.711,A -85,B 0,C 180,E1 -12197.558,E2 -12197.558} C_VEL
LIN {X 0,Y 374.934,Z 454.364,A -85,B 0,C 180,E1 -12199.311,E2 -12199.311} C_VEL
LIN {X 0,Y 379.078,Z 469.157,A -85,B 0,C 180,E1 -12200.073,E2 -12200.073} C_VEL
LIN {X 0,Y 382.653,Z 482.828,A -85,B 0,C 180,E1 -12200.964,E2 -12200.964} C_VEL
LIN {X 0,Y 383.218,Z 485.389,A -85,B 0,C 180,E1 -12201.149,E2 -12201.149} C_VEL
LIN {X 0,Y 382.413,Z 498.001,A -85,B 0,C 180,E1 -12202.004,E2 -12202.004} C_VEL
LIN {X 0,Y 381.362,Z 510.32,A -85,B 0,C 180,E1 -12203.041,E2 -12203.041} C_VEL
LIN {X 0,Y 380.206,Z 522.561,A -85,B 0,C 180,E1 -12204.311,E2 -12204.311} C_VEL
LIN {X 0,Y 379.067,Z 533.742,A -85,B 0,C 180,E1 -12205.725,E2 -12205.725} C_VEL
LIN {X 0,Y 377.979,Z 544.441,A -85,B 0,C 180,E1 -12207.369,E2 -12207.369} C_VEL
LIN {X 0,Y 376.935,Z 553.447,A -85,B 0,C 180,E1 -12209.055,E2 -12209.055} C_VEL
LIN {X 0,Y 376.18,Z 561.62,A -85,B 0,C 180,E1 -12210.938,E2 -12210.938} C_VEL
LIN {X 0,Y 375.617,Z 567.889,A -85,B 0,C 180,E1 -12212.715,E2 -12212.715} C_VEL
LIN {X 0,Y 375.2,Z 572.905,A -85,B 0,C 180,E1 -12214.48,E2 -12214.48} C_VEL
LIN {X 0,Y 374.877,Z 576.785,A -85,B 0,C 180,E1 -12216.23,E2 -12216.23} C_VEL
LIN {X 0,Y 374.623,Z 579.623,A -85,B 0,C 180,E1 -12217.963,E2 -12217.963} C_VEL
LIN {X 0,Y 374.533,Z 582.019,A -85,B 0,C 180,E1 -12220.259,E2 -12220.259} C_VEL
LIN {X 0,Y 374.499,Z 582.625,A -85,B 0,C 180,E1 -12221.395,E2 -12221.395} C_VEL
LIN {X 0,Y 374.532,Z 582.68,A -85,B 0,C 180,E1 -12223.652,E2 -12223.652} C_VEL
LIN {X 0,Y 374.693,Z 581.282,A -85,B 0,C 180,E1 -12225.887,E2 -12225.887} C_VEL
LIN {X 0,Y 375.081,Z 578.437,A -85,B 0,C 180,E1 -12228.105,E2 -12228.105} C_VEL
LIN {X 0,Y 375.583,Z 574.118,A -85,B 0,C 180,E1 -12230.304,E2 -12230.304} C_VEL
LIN {X 0,Y 376.125,Z 569.602,A -85,B 0,C 180,E1 -12232.013,E2 -12232.013} C_VEL
LIN {X 0,Y 377.081,Z 562.577,A -85,B 0,C 180,E1 -12234.116,E2 -12234.116} C_VEL
LIN {X 0,Y 378.271,Z 554.542,A -85,B 0,C 180,E1 -12236.005,E2 -12236.005} C_VEL
LIN {X 0,Y 379.307,Z 546.264,A -85,B 0,C 180,E1 -12237.61,E2 -12237.61} C_VEL
LIN {X 0,Y 380.722,Z 536.225,A -85,B 0,C 180,E1 -12239.207,E2 -12239.207} C_VEL
LIN {X 0,Y 382.315,Z 524.1,A -85,B 0,C 180,E1 -12240.79,E2 -12240.79} C_VEL
LIN {X 0,Y 383.844,Z 511.728,A -85,B 0,C 180,E1 -12242.098,E2 -12242.098} C_VEL
LIN {X 0,Y 385.142,Z 499.583,A -85,B 0,C 180,E1 -12243.138,E2 -12243.138} C_VEL
LIN {X 0,Y 386.082,Z 489.901,A -85,B 0,C 180,E1 -12243.81,E2 -12243.81} C_VEL
LIN {X 0,Y 384.783,Z 483.885,A -85,B 0,C 180,E1 -12244.321,E2 -12244.321} C_VEL
LIN {X 0,Y 380.421,Z 470.123,A -85,B 0,C 180,E1 -12245.479,E2 -12245.479} C_VEL
LIN {X 0,Y 376.73,Z 461.524,A -85,B 0,C 180,E1 -12246.189,E2 -12246.189} C_VEL
LIN {X 0,Y 375.827,Z 458.864,A -85,B 0,C 180,E1 -12246.375,E2 -12246.375} C_VEL
LIN {X 0,Y 375.92,Z 457.488,A -85,B 0,C 180,E1 -12248.601,E2 -12248.601} C_VEL
LIN {X 0,Y 376.045,Z 455.625,A -85,B 0,C 180,E1 -12251.863,E2 -12251.863} C_VEL
LIN {X 0,Y 376.225,Z 453.92,A -85,B 0,C 180,E1 -12255.16,E2 -12255.16} C_VEL
LIN {X 0,Y 376.466,Z 452.428,A -85,B 0,C 180,E1 -12258.503,E2 -12258.503} C_VEL
LIN {X 0,Y 376.558,Z 451.517,A -85,B 0,C 180,E1 -12261.065,E2 -12261.065} C_VEL
LIN {X 0,Y 376.509,Z 450.677,A -85,B 0,C 180,E1 -12264.246,E2 -12264.246} C_VEL
LIN {X 0,Y 376.487,Z 450.203,A -85,B 0,C 180,E1 -12267.819,E2 -12267.819} C_VEL
LIN {X 0,Y 376.485,Z 450.335,A -85,B 0,C 180,E1 -12271.513,E2 -12271.513} C_VEL
LIN {X 0,Y 376.608,Z 451.08,A -85,B 0,C 180,E1 -12274.807,E2 -12274.807} C_VEL
LIN {X 0,Y 376.938,Z 452.629,A -85,B 0,C 180,E1 -12278.457,E2 -12278.457} C_VEL
LIN {X 0,Y 377.378,Z 455.078,A -85,B 0,C 180,E1 -12282.101,E2 -12282.101} C_VEL
LIN {X 0,Y 377.807,Z 457.66,A -85,B 0,C 180,E1 -12285.019,E2 -12285.019} C_VEL
LIN {X 0,Y 378.337,Z 460.923,A -85,B 0,C 180,E1 -12288.031,E2 -12288.031} C_VEL
LIN {X 0,Y 378.558,Z 462.838,A -85,B 0,C 180,E1 -12289.568,E2 -12289.568} C_VEL
LIN {X 0,Y 378.452,Z 466.54,A -85,B 0,C 180,E1 -12292.207,E2 -12292.207} C_VEL
LIN {X 0,Y 377.741,Z 470.885,A -85,B 0,C 180,E1 -12294.948,E2 -12294.948} C_VEL
LIN {X 0,Y 376.95,Z 477.13,A -85,B 0,C 180,E1 -12298.531,E2 -12298.531} C_VEL
LIN {X 0,Y 376.407,Z 482.408,A -85,B 0,C 180,E1 -12301.348,E2 -12301.348} C_VEL
LIN {X 0,Y 375.838,Z 488.696,A -85,B 0,C 180,E1 -12304.527,E2 -12304.527} C_VEL
LIN {X 0,Y 375.679,Z 490.777,A -85,B 0,C 180,E1 -12305.55,E2 -12305.55} C_VEL
LIN {X 0,Y 376.614,Z 494.332,A -85,B 0,C 180,E1 -12305.762,E2 -12305.762} C_VEL
LIN {X 0,Y 380.241,Z 508.254,A -85,B 0,C 180,E1 -12306.658,E2 -12306.658} C_VEL
LIN {X 0,Y 382.577,Z 522.629,A -85,B 0,C 180,E1 -12307.641,E2 -12307.641} C_VEL
LIN {X 0,Y 383.637,Z 535.972,A -85,B 0,C 180,E1 -12308.662,E2 -12308.662} C_VEL
LIN {X 0,Y 382.845,Z 544.825,A -85,B 0,C 180,E1 -12309.36,E2 -12309.36} C_VEL
LIN {X 0,Y 381.472,Z 556.376,A -85,B 0,C 180,E1 -12310.421,E2 -12310.421} C_VEL
LIN {X 0,Y 379.878,Z 568.83,A -85,B 0,C 180,E1 -12311.809,E2 -12311.809} C_VEL
LIN {X 0,Y 378.477,Z 579.664,A -85,B 0,C 180,E1 -12313.273,E2 -12313.273} C_VEL
LIN {X 0,Y 377.258,Z 589.551,A -85,B 0,C 180,E1 -12314.882,E2 -12314.882} C_VEL
LIN {X 0,Y 376.407,Z 598.025,A -85,B 0,C 180,E1 -12316.543,E2 -12316.543} C_VEL
LIN {X 0,Y 375.592,Z 605.873,A -85,B 0,C 180,E1 -12318.396,E2 -12318.396} C_VEL
LIN {X 0,Y 375.028,Z 612.386,A -85,B 0,C 180,E1 -12320.29,E2 -12320.29} C_VEL
LIN {X 0,Y 374.721,Z 618.203,A -85,B 0,C 180,E1 -12322.456,E2 -12322.456} C_VEL
LIN {X 0,Y 374.637,Z 621.063,A -85,B 0,C 180,E1 -12323.854,E2 -12323.854} C_VEL
LIN {X 0,Y 374.582,Z 623.93,A -85,B 0,C 180,E1 -12325.696,E2 -12325.696} C_VEL
LIN {X 0,Y 374.684,Z 625.938,A -85,B 0,C 180,E1 -12327.85,E2 -12327.85} C_VEL
LIN {X 0,Y 374.653,Z 626.534,A -85,B 0,C 180,E1 -12330,E2 -12330} C_VEL
LIN {X 0,Y 374.704,Z 625.727,A -85,B 0,C 180,E1 -12332.15,E2 -12332.15} C_VEL
LIN {X 0,Y 374.577,Z 623.483,A -85,B 0,C 180,E1 -12334.304,E2 -12334.304} C_VEL
LIN {X 0,Y 374.676,Z 619.771,A -85,B 0,C 180,E1 -12336.462,E2 -12336.462} C_VEL
LIN {X 0,Y 374.832,Z 614.461,A -85,B 0,C 180,E1 -12338.627,E2 -12338.627} C_VEL
LIN {X 0,Y 375.134,Z 609.292,A -85,B 0,C 180,E1 -12340.252,E2 -12340.252} C_VEL
LIN {X 0,Y 375.728,Z 601.9,A -85,B 0,C 180,E1 -12342.147,E2 -12342.147} C_VEL
LIN {X 0,Y 376.424,Z 593.664,A -85,B 0,C 180,E1 -12343.865,E2 -12343.865} C_VEL
LIN {X 0,Y 377.498,Z 583.082,A -85,B 0,C 180,E1 -12345.661,E2 -12345.661} C_VEL
LIN {X 0,Y 378.551,Z 572.461,A -85,B 0,C 180,E1 -12347.141,E2 -12347.141} C_VEL
LIN {X 0,Y 379.919,Z 560.841,A -85,B 0,C 180,E1 -12348.469,E2 -12348.469} C_VEL
LIN {X 0,Y 380.991,Z 549.437,A -85,B 0,C 180,E1 -12349.545,E2 -12349.545} C_VEL
LIN {X 0,Y 382.192,Z 535.948,A -85,B 0,C 180,E1 -12350.57,E2 -12350.57} C_VEL
LIN {X 0,Y 380.467,Z 522.599,A -85,B 0,C 180,E1 -12351.483,E2 -12351.483} C_VEL
LIN {X 0,Y 378.069,Z 508.016,A -85,B 0,C 180,E1 -12352.284,E2 -12352.284} C_VEL
LIN {X 0,Y 375.585,Z 494.973,A -85,B 0,C 180,E1 -12352.846,E2 -12352.846} C_VEL
LIN {X 0,Y 376.173,Z 487.067,A -85,B 0,C 180,E1 -12356.64,E2 -12356.64} C_VEL
LIN {X 0,Y 376.77,Z 479.726,A -85,B 0,C 180,E1 -12360.24,E2 -12360.24} C_VEL
LIN {X 0,Y 377.339,Z 474.147,A -85,B 0,C 180,E1 -12363.057,E2 -12363.057} C_VEL
LIN {X 0,Y 377.963,Z 467.497,A -85,B 0,C 180,E1 -12366.513,E2 -12366.513} C_VEL
LIN {X 0,Y 378.418,Z 462.579,A -85,B 0,C 180,E1 -12369.156,E2 -12369.156} C_VEL
LIN {X 0,Y 378.082,Z 458.932,A -85,B 0,C 180,E1 -12371.24,E2 -12371.24} C_VEL
LIN {X 0,Y 376.991,Z 452.9,A -85,B 0,C 180,E1 -12374.894,E2 -12374.894} C_VEL
LIN {X 0,Y 376.011,Z 447.271,A -85,B 0,C 180,E1 -12378.571,E2 -12378.571} C_VEL
LIN {X 0,Y 375.96,Z 447.282,A -85,B 0,C 180,E1 -12381.911,E2 -12381.911} C_VEL
LIN {X 0,Y 375.975,Z 447.279,A -85,B 0,C 180,E1 -12385.332,E2 -12385.332} C_VEL
LIN {X 0,Y 375.972,Z 447.276,A -85,B 0,C 180,E1 -12388.439,E2 -12388.439} C_VEL
LIN {X 0,Y 375.997,Z 447.272,A -85,B 0,C 180,E1 -12392.142,E2 -12392.142} C_VEL
LIN {X 0,Y 376.001,Z 447.274,A -85,B 0,C 180,E1 -12394.539,E2 -12394.539} C_VEL
LIN {X 0,Y 375.957,Z 447.277,A -85,B 0,C 180,E1 -12398.046,E2 -12398.046} C_VEL
LIN {X 0,Y 376.003,Z 447.272,A -85,B 0,C 180,E1 -12401.473,E2 -12401.473} C_VEL
LIN {X 0,Y 376.052,Z 447.27,A -85,B 0,C 180,E1 -12404.832,E2 -12404.832} C_VEL
LIN {X 0,Y 376.045,Z 447.267,A -85,B 0,C 180,E1 -12408.137,E2 -12408.137} C_VEL
LIN {X 0,Y 376.252,Z 447.241,A -85,B 0,C 180,E1 -12411.877,E2 -12411.877} C_VEL
LIN {X 0,Y 376.167,Z 447.255,A -85,B 0,C 180,E1 -12414.64,E2 -12414.64} C_VEL
LIN {X 0,Y 376.348,Z 447.229,A -85,B 0,C 180,E1 -12417.86,E2 -12417.86} C_VEL
LIN {X 0,Y 376.483,Z 447.212,A -85,B 0,C 180,E1 -12420,E2 -12420} C_VEL
LIN {X 0,Y 376.186,Z 447.249,A -85,B 0,C 180,E1 -12423.213,E2 -12423.213} C_VEL
LIN {X 0,Y 376.239,Z 447.245,A -85,B 0,C 180,E1 -12426.567,E2 -12426.567} C_VEL
LIN {X 0,Y 376.2,Z 447.251,A -85,B 0,C 180,E1 -12428.595,E2 -12428.595} C_VEL
LIN {X 0,Y 376.044,Z 447.268,A -85,B 0,C 180,E1 -12431.864,E2 -12431.864} C_VEL
LIN {X 0,Y 376.053,Z 447.266,A -85,B 0,C 180,E1 -12435.168,E2 -12435.168} C_VEL
LIN {X 0,Y 376.019,Z 447.273,A -85,B 0,C 180,E1 -12438.527,E2 -12438.527} C_VEL
LIN {X 0,Y 375.959,Z 447.28,A -85,B 0,C 180,E1 -12441.955,E2 -12441.955} C_VEL
LIN {X 0,Y 376.002,Z 447.272,A -85,B 0,C 180,E1 -12445.462,E2 -12445.462} C_VEL
LIN {X 0,Y 375.966,Z 447.276,A -85,B 0,C 180,E1 -12449.08,E2 -12449.08} C_VEL
LIN {X 0,Y 375.946,Z 447.28,A -85,B 0,C 180,E1 -12452.829,E2 -12452.829} C_VEL
LIN {X 0,Y 375.955,Z 447.278,A -85,B 0,C 180,E1 -12455.416,E2 -12455.416} C_VEL
LIN {X 0,Y 375.972,Z 447.279,A -85,B 0,C 180,E1 -12458.271,E2 -12458.271} C_VEL
LIN {X 0,Y 375.933,Z 447.282,A -85,B 0,C 180,E1 -12461.602,E2 -12461.602} C_VEL
LIN {X 0,Y 375.927,Z 447.281,A -85,B 0,C 180,E1 -12465.269,E2 -12465.269} C_VEL
LIN {X 0,Y 375.959,Z 447.279,A -85,B 0,C 180,E1 -12468.396,E2 -12468.396} C_VEL
LIN {X 0,Y 375.978,Z 447.279,A -85,B 0,C 180,E1 -12471.73,E2 -12471.73} C_VEL
LIN {X 0,Y 375.98,Z 447.276,A -85,B 0,C 180,E1 -12475.333,E2 -12475.333} C_VEL
LIN {X 0,Y 375.961,Z 447.277,A -85,B 0,C 180,E1 -12478.439,E2 -12478.439} C_VEL
LIN {X 0,Y 376.004,Z 447.274,A -85,B 0,C 180,E1 -12482.143,E2 -12482.143} C_VEL
LIN {X 0,Y 376.008,Z 447.271,A -85,B 0,C 180,E1 -12484.54,E2 -12484.54} C_VEL
LIN {X 0,Y 375.966,Z 447.279,A -85,B 0,C 180,E1 -12488.046,E2 -12488.046} C_VEL
LIN {X 0,Y 376.027,Z 447.272,A -85,B 0,C 180,E1 -12491.474,E2 -12491.474} C_VEL
LIN {X 0,Y 376.062,Z 447.265,A -85,B 0,C 180,E1 -12494.833,E2 -12494.833} C_VEL
LIN {X 0,Y 376.053,Z 447.267,A -85,B 0,C 180,E1 -12498.137,E2 -12498.137} C_VEL
LIN {X 0,Y 376.197,Z 447.25,A -85,B 0,C 180,E1 -12501.947,E2 -12501.947} C_VEL
LIN {X 0,Y 376.164,Z 447.252,A -85,B 0,C 180,E1 -12504.64,E2 -12504.64} C_VEL
LIN {X 0,Y 376.358,Z 447.23,A -85,B 0,C 180,E1 -12507.86,E2 -12507.86} C_VEL
LIN {X 0,Y 376.491,Z 447.211,A -85,B 0,C 180,E1 -12510,E2 -12510} C_VEL
LIN {X 0,Y 376.189,Z 447.252,A -85,B 0,C 180,E1 -12513.213,E2 -12513.213} C_VEL
LIN {X 0,Y 376.24,Z 447.242,A -85,B 0,C 180,E1 -12516.435,E2 -12516.435} C_VEL
LIN {X 0,Y 376.122,Z 447.259,A -85,B 0,C 180,E1 -12519.681,E2 -12519.681} C_VEL
LIN {X 0,Y 376.093,Z 447.262,A -85,B 0,C 180,E1 -12523.657,E2 -12523.657} C_VEL
LIN {X 0,Y 376.046,Z 447.268,A -85,B 0,C 180,E1 -12527.607,E2 -12527.607} C_VEL
LIN {X 0,Y 375.98,Z 447.278,A -85,B 0,C 180,E1 -12530.832,E2 -12530.832} C_VEL
LIN {X 0,Y 375.996,Z 447.273,A -85,B 0,C 180,E1 -12534.281,E2 -12534.281} C_VEL
LIN {X 0,Y 376.021,Z 447.272,A -85,B 0,C 180,E1 -12536.651,E2 -12536.651} C_VEL
LIN {X 0,Y 375.972,Z 447.279,A -85,B 0,C 180,E1 -12539.078,E2 -12539.078} C_VEL
LIN {X 0,Y 375.937,Z 447.284,A -85,B 0,C 180,E1 -12542.829,E2 -12542.829} C_VEL
LIN {X 0,Y 375.83,Z 447.295,A -85,B 0,C 180,E1 -12545.429,E2 -12545.429} C_VEL
LIN {X 0,Y 375.469,Z 447.339,A -85,B 0,C 180,E1 -12548.172,E2 -12548.172} C_VEL
LIN {X 0,Y 375.256,Z 447.37,A -85,B 0,C 180,E1 -12550.019,E2 -12550.019} C_VEL
LIN {X 0,Y 374.459,Z 447.597,A -85,B 0,C 180,E1 -12550.911,E2 -12550.911} C_VEL
LIN {X 0,Y 371.473,Z 448.658,A -85,B 0,C 180,E1 -12552.352,E2 -12552.352} C_VEL
LIN {X 0,Y 369.027,Z 449.828,A -85,B 0,C 180,E1 -12553.515,E2 -12553.515} C_VEL
LIN {X 0,Y 368.012,Z 450.697,A -85,B 0,C 180,E1 -12554.415,E2 -12554.415} C_VEL
LIN {X 0,Y 367.945,Z 450.965,A -85,B 0,C 180,E1 -12554.721,E2 -12554.721} C_VEL
LIN {X 0,Y 367.828,Z 454.312,A -85,B 0,C 180,E1 -12558.559,E2 -12558.559} C_VEL
LIN {X 0,Y 367.834,Z 454.764,A -85,B 0,C 180,E1 -12558.933,E2 -12558.933} C_VEL
LIN {X 0,Y 372.145,Z 469.773,A -85,B 0,C 180,E1 -12559.737,E2 -12559.737} C_VEL
LIN {X 0,Y 375.686,Z 483.659,A -85,B 0,C 180,E1 -12560.666,E2 -12560.666} C_VEL
LIN {X 0,Y 376.454,Z 487.504,A -85,B 0,C 180,E1 -12560.954,E2 -12560.954} C_VEL
LIN {X 0,Y 375.377,Z 501.147,A -85,B 0,C 180,E1 -12561.928,E2 -12561.928} C_VEL
LIN {X 0,Y 374.263,Z 513.781,A -85,B 0,C 180,E1 -12563.065,E2 -12563.065} C_VEL
LIN {X 0,Y 373.002,Z 526.036,A -85,B 0,C 180,E1 -12564.427,E2 -12564.427} C_VEL
LIN {X 0,Y 371.81,Z 537.305,A -85,B 0,C 180,E1 -12565.964,E2 -12565.964} C_VEL
LIN {X 0,Y 370.759,Z 547.309,A -85,B 0,C 180,E1 -12567.622,E2 -12567.622} C_VEL
LIN {X 0,Y 369.667,Z 556.317,A -85,B 0,C 180,E1 -12569.431,E2 -12569.431} C_VEL
LIN {X 0,Y 369.029,Z 563.367,A -85,B 0,C 180,E1 -12571.168,E2 -12571.168} C_VEL
LIN {X 0,Y 368.359,Z 570.397,A -85,B 0,C 180,E1 -12573.313,E2 -12573.313} C_VEL
LIN {X 0,Y 367.984,Z 575.052,A -85,B 0,C 180,E1 -12575.154,E2 -12575.154} C_VEL
LIN {X 0,Y 367.768,Z 577.799,A -85,B 0,C 180,E1 -12576.528,E2 -12576.528} C_VEL
LIN {X 0,Y 367.494,Z 580.96,A -85,B 0,C 180,E1 -12578.693,E2 -12578.693} C_VEL
LIN {X 0,Y 367.481,Z 582.095,A -85,B 0,C 180,E1 -12579.864,E2 -12579.864} C_VEL
LIN {X 0,Y 367.404,Z 583.219,A -85,B 0,C 180,E1 -12582.178,E2 -12582.178} C_VEL
LIN {X 0,Y 367.48,Z 582.857,A -85,B 0,C 180,E1 -12584.469,E2 -12584.469} C_VEL
LIN {X 0,Y 367.764,Z 581.01,A -85,B 0,C 180,E1 -12586.743,E2 -12586.743} C_VEL
LIN {X 0,Y 368.198,Z 577.702,A -85,B 0,C 180,E1 -12588.996,E2 -12588.996} C_VEL
LIN {X 0,Y 368.844,Z 572.891,A -85,B 0,C 180,E1 -12591.232,E2 -12591.232} C_VEL
LIN {X 0,Y 369.483,Z 568.217,A -85,B 0,C 180,E1 -12592.898,E2 -12592.898} C_VEL
LIN {X 0,Y 370.484,Z 561.443,A -85,B 0,C 180,E1 -12594.83,E2 -12594.83} C_VEL
LIN {X 0,Y 371.705,Z 553.079,A -85,B 0,C 180,E1 -12596.748,E2 -12596.748} C_VEL
LIN {X 0,Y 373.007,Z 544.255,A -85,B 0,C 180,E1 -12598.411,E2 -12598.411} C_VEL
LIN {X 0,Y 374.511,Z 534.036,A -85,B 0,C 180,E1 -12600,E2 -12600} C_VEL
LIN {X 0,Y 376.111,Z 522.468,A -85,B 0,C 180,E1 -12601.472,E2 -12601.472} C_VEL
LIN {X 0,Y 377.72,Z 509.532,A -85,B 0,C 180,E1 -12602.799,E2 -12602.799} C_VEL
LIN {X 0,Y 379.129,Z 496.804,A -85,B 0,C 180,E1 -12603.853,E2 -12603.853} C_VEL
LIN {X 0,Y 379.697,Z 491.199,A -85,B 0,C 180,E1 -12604.246,E2 -12604.246} C_VEL
LIN {X 0,Y 376.858,Z 480.342,A -85,B 0,C 180,E1 -12605.237,E2 -12605.237} C_VEL
LIN {X 0,Y 372.703,Z 468.551,A -85,B 0,C 180,E1 -12606.272,E2 -12606.272} C_VEL
LIN {X 0,Y 368.984,Z 460.199,A -85,B 0,C 180,E1 -12607.007,E2 -12607.007} C_VEL
LIN {X 0,Y 368.847,Z 459.466,A -85,B 0,C 180,E1 -12607.092,E2 -12607.092} C_VEL
LIN {X 0,Y 368.942,Z 457.841,A -85,B 0,C 180,E1 -12609.871,E2 -12609.871} C_VEL
LIN {X 0,Y 369.184,Z 455.727,A -85,B 0,C 180,E1 -12613.869,E2 -12613.869} C_VEL
LIN {X 0,Y 369.45,Z 453.888,A -85,B 0,C 180,E1 -12617.987,E2 -12617.987} C_VEL
LIN {X 0,Y 369.57,Z 452.747,A -85,B 0,C 180,E1 -12621.283,E2 -12621.283} C_VEL
LIN {X 0,Y 369.524,Z 451.962,A -85,B 0,C 180,E1 -12624.735,E2 -12624.735} C_VEL
LIN {X 0,Y 369.533,Z 451.684,A -85,B 0,C 180,E1 -12627.158,E2 -12627.158} C_VEL
LIN {X 0,Y 369.532,Z 451.65,A -85,B 0,C 180,E1 -12629.636,E2 -12629.636} C_VEL
LIN {X 0,Y 369.621,Z 452.23,A -85,B 0,C 180,E1 -12633.464,E2 -12633.464} C_VEL
LIN {X 0,Y 369.846,Z 453.48,A -85,B 0,C 180,E1 -12637.052,E2 -12637.052} C_VEL
LIN {X 0,Y 370.19,Z 455.232,A -85,B 0,C 180,E1 -12640.202,E2 -12640.202} C_VEL
LIN {X 0,Y 370.552,Z 457.369,A -85,B 0,C 180,E1 -12643.062,E2 -12643.062} C_VEL
LIN {X 0,Y 371.017,Z 460.162,A -85,B 0,C 180,E1 -12646.039,E2 -12646.039} C_VEL
LIN {X 0,Y 371.522,Z 463.723,A -85,B 0,C 180,E1 -12649.172,E2 -12649.172} C_VEL
LIN {X 0,Y 371.544,Z 466.632,A -85,B 0,C 180,E1 -12651.376,E2 -12651.376} C_VEL
LIN {X 0,Y 370.957,Z 470.64,A -85,B 0,C 180,E1 -12654.034,E2 -12654.034} C_VEL
LIN {X 0,Y 370.215,Z 475.951,A -85,B 0,C 180,E1 -12657.247,E2 -12657.247} C_VEL
LIN {X 0,Y 369.583,Z 481.509,A -85,B 0,C 180,E1 -12660.369,E2 -12660.369} C_VEL
LIN {X 0,Y 368.874,Z 488.469,A -85,B 0,C 180,E1 -12664.011,E2 -12664.011} C_VEL
LIN {X 0,Y 368.731,Z 490.292,A -85,B 0,C 180,E1 -12664.889,E2 -12664.889} C_VEL
LIN {X 0,Y 369.639,Z 493.69,A -85,B 0,C 180,E1 -12665.103,E2 -12665.103} C_VEL
LIN {X 0,Y 373.473,Z 507.813,A -85,B 0,C 180,E1 -12666.069,E2 -12666.069} C_VEL
LIN {X 0,Y 375.708,Z 520.562,A -85,B 0,C 180,E1 -12666.987,E2 -12666.987} C_VEL
LIN {X 0,Y 376.912,Z 534.768,A -85,B 0,C 180,E1 -12668.104,E2 -12668.104} C_VEL
LIN {X 0,Y 376.932,Z 539.938,A -85,B 0,C 180,E1 -12668.537,E2 -12668.537} C_VEL
LIN {X 0,Y 375.171,Z 553.38,A -85,B 0,C 180,E1 -12669.715,E2 -12669.715} C_VEL
LIN {X 0,Y 373.594,Z 565.753,A -85,B 0,C 180,E1 -12671.065,E2 -12671.065} C_VEL
LIN {X 0,Y 372.17,Z 576.011,A -85,B 0,C 180,E1 -12672.414,E2 -12672.414} C_VEL
LIN {X 0,Y 370.777,Z 586.429,A -85,B 0,C 180,E1 -12674.048,E2 -12674.048} C_VEL
LIN {X 0,Y 369.558,Z 596.135,A -85,B 0,C 180,E1 -12675.902,E2 -12675.902} C_VEL
LIN {X 0,Y 368.703,Z 604.619,A -85,B 0,C 180,E1 -12677.897,E2 -12677.897} C_VEL
LIN {X 0,Y 368.101,Z 610.418,A -85,B 0,C 180,E1 -12679.55,E2 -12679.55} C_VEL
LIN {X 0,Y 367.693,Z 616.566,A -85,B 0,C 180,E1 -12681.758,E2 -12681.758} C_VEL
LIN {X 0,Y 367.534,Z 621.017,A -85,B 0,C 180,E1 -12683.904,E2 -12683.904} C_VEL
LIN {X 0,Y 367.509,Z 623.557,A -85,B 0,C 180,E1 -12685.613,E2 -12685.613} C_VEL
LIN {X 0,Y 367.583,Z 625.532,A -85,B 0,C 180,E1 -12687.809,E2 -12687.809} C_VEL
LIN {X 0,Y 367.584,Z 626.097,A -85,B 0,C 180,E1 -12690,E2 -12690} C_VEL
LIN {X 0,Y 367.617,Z 625.255,A -85,B 0,C 180,E1 -12692.191,E2 -12692.191} C_VEL
LIN {X 0,Y 367.506,Z 622.978,A -85,B 0,C 180,E1 -12694.387,E2 -12694.387} C_VEL
LIN {X 0,Y 367.589,Z 619.225,A -85,B 0,C 180,E1 -12696.587,E2 -12696.587} C_VEL
LIN {X 0,Y 367.714,Z 615.33,A -85,B 0,C 180,E1 -12698.241,E2 -12698.241} C_VEL
LIN {X 0,Y 367.968,Z 610.493,A -85,B 0,C 180,E1 -12699.898,E2 -12699.898} C_VEL
LIN {X 0,Y 368.555,Z 603.476,A -85,B 0,C 180,E1 -12701.829,E2 -12701.829} C_VEL
LIN {X 0,Y 369.164,Z 596.269,A -85,B 0,C 180,E1 -12703.456,E2 -12703.456} C_VEL
LIN {X 0,Y 370.017,Z 587.283,A -85,B 0,C 180,E1 -12705.139,E2 -12705.139} C_VEL
LIN {X 0,Y 371.216,Z 576.625,A -85,B 0,C 180,E1 -12706.781,E2 -12706.781} C_VEL
LIN {X 0,Y 372.333,Z 565.913,A -85,B 0,C 180,E1 -12708.146,E2 -12708.146} C_VEL
LIN {X 0,Y 373.604,Z 554.338,A -85,B 0,C 180,E1 -12709.363,E2 -12709.363} C_VEL
LIN {X 0,Y 374.879,Z 541.31,A -85,B 0,C 180,E1 -12710.474,E2 -12710.474} C_VEL
LIN {X 0,Y 375.23,Z 536.197,A -85,B 0,C 180,E1 -12710.846,E2 -12710.846} C_VEL
LIN {X 0,Y 373.419,Z 521.924,A -85,B 0,C 180,E1 -12711.842,E2 -12711.842} C_VEL
LIN {X 0,Y 370.819,Z 506.809,A -85,B 0,C 180,E1 -12712.683,E2 -12712.683} C_VEL
LIN {X 0,Y 368.53,Z 494.597,A -85,B 0,C 180,E1 -12713.24,E2 -12713.24} C_VEL
LIN {X 0,Y 369.057,Z 487.98,A -85,B 0,C 180,E1 -12716.488,E2 -12716.488} C_VEL
LIN {X 0,Y 369.726,Z 480.493,A -85,B 0,C 180,E1 -12720.246,E2 -12720.246} C_VEL
LIN {X 0,Y 370.453,Z 473.156,A -85,B 0,C 180,E1 -12724.031,E2 -12724.031} C_VEL
LIN {X 0,Y 371.14,Z 467.024,A -85,B 0,C 180,E1 -12727.314,E2 -12727.314} C_VEL
LIN {X 0,Y 371.399,Z 463.751,A -85,B 0,C 180,E1 -12729.118,E2 -12729.118} C_VEL
LIN {X 0,Y 370.997,Z 459.613,A -85,B 0,C 180,E1 -12731.53,E2 -12731.53} C_VEL
LIN {X 0,Y 369.889,Z 453.479,A -85,B 0,C 180,E1 -12735.331,E2 -12735.331} C_VEL
LIN {X 0,Y 368.962,Z 448.15,A -85,B 0,C 180,E1 -12738.917,E2 -12738.917} C_VEL
LIN {X 0,Y 368.9,Z 448.16,A -85,B 0,C 180,E1 -12742.437,E2 -12742.437} C_VEL
LIN {X 0,Y 368.932,Z 448.156,A -85,B 0,C 180,E1 -12745.146,E2 -12745.146} C_VEL
LIN {X 0,Y 368.924,Z 448.158,A -85,B 0,C 180,E1 -12749.046,E2 -12749.046} C_VEL
LIN {X 0,Y 368.982,Z 448.147,A -85,B 0,C 180,E1 -12751.564,E2 -12751.564} C_VEL
LIN {X 0,Y 368.952,Z 448.153,A -85,B 0,C 180,E1 -12755.224,E2 -12755.224} C_VEL
LIN {X 0,Y 368.932,Z 448.156,A -85,B 0,C 180,E1 -12758.973,E2 -12758.973} C_VEL
LIN {X 0,Y 368.985,Z 448.146,A -85,B 0,C 180,E1 -12762.257,E2 -12762.257} C_VEL
LIN {X 0,Y 369.031,Z 448.141,A -85,B 0,C 180,E1 -12766.228,E2 -12766.228} C_VEL
LIN {X 0,Y 369.062,Z 448.137,A -85,B 0,C 180,E1 -12770.132,E2 -12770.132} C_VEL
LIN {X 0,Y 369.182,Z 448.124,A -85,B 0,C 180,E1 -12772.342,E2 -12772.342} C_VEL
LIN {X 0,Y 369.139,Z 448.13,A -85,B 0,C 180,E1 -12774.538,E2 -12774.538} C_VEL
LIN {X 0,Y 369.313,Z 448.105,A -85,B 0,C 180,E1 -12777.819,E2 -12777.819} C_VEL
LIN {X 0,Y 369.452,Z 448.088,A -85,B 0,C 180,E1 -12780,E2 -12780} C_VEL
LIN {X 0,Y 369.314,Z 448.107,A -85,B 0,C 180,E1 -12782.181,E2 -12782.181} C_VEL
LIN {X 0,Y 369.209,Z 448.122,A -85,B 0,C 180,E1 -12786.558,E2 -12786.558} C_VEL
LIN {X 0,Y 369.132,Z 448.13,A -85,B 0,C 180,E1 -12788.761,E2 -12788.761} C_VEL
LIN {X 0,Y 369,Z 448.147,A -85,B 0,C 180,E1 -12792.094,E2 -12792.094} C_VEL
LIN {X 0,Y 368.992,Z 448.145,A -85,B 0,C 180,E1 -12795.465,E2 -12795.465} C_VEL
LIN {X 0,Y 368.977,Z 448.148,A -85,B 0,C 180,E1 -12798.893,E2 -12798.893} C_VEL
LIN {X 0,Y 368.928,Z 448.157,A -85,B 0,C 180,E1 -12802.396,E2 -12802.396} C_VEL
LIN {X 0,Y 368.996,Z 448.148,A -85,B 0,C 180,E1 -12805.981,E2 -12805.981} C_VEL
LIN {X 0,Y 368.955,Z 448.151,A -85,B 0,C 180,E1 -12808.812,E2 -12808.812} C_VEL
LIN {X 0,Y 368.895,Z 448.161,A -85,B 0,C 180,E1 -12812.239,E2 -12812.239} C_VEL
LIN {X 0,Y 368.926,Z 448.153,A -85,B 0,C 180,E1 -12815.002,E2 -12815.002} C_VEL
LIN {X 0,Y 368.907,Z 448.157,A -85,B 0,C 180,E1 -12818.641,E2 -12818.641} C_VEL
LIN {X 0,Y 368.88,Z 448.163,A -85,B 0,C 180,E1 -12822.01,E2 -12822.01} C_VEL
LIN {X 0,Y 368.88,Z 448.158,A -85,B 0,C 180,E1 -12825.177,E2 -12825.177} C_VEL
LIN {X 0,Y 368.909,Z 448.159,A -85,B 0,C 180,E1 -12828.182,E2 -12828.182} C_VEL
LIN {X 0,Y 368.913,Z 448.156,A -85,B 0,C 180,E1 -12831.36,E2 -12831.36} C_VEL
LIN {X 0,Y 368.937,Z 448.152,A -85,B 0,C 180,E1 -12835.147,E2 -12835.147} C_VEL
LIN {X 0,Y 368.93,Z 448.152,A -85,B 0,C 180,E1 -12839.047,E2 -12839.047} C_VEL
LIN {X 0,Y 368.988,Z 448.149,A -85,B 0,C 180,E1 -12841.565,E2 -12841.565} C_VEL
LIN {X 0,Y 368.96,Z 448.15,A -85,B 0,C 180,E1 -12845.225,E2 -12845.225} C_VEL
LIN {X 0,Y 368.94,Z 448.152,A -85,B 0,C 180,E1 -12848.974,E2 -12848.974} C_VEL
LIN {X 0,Y 368.993,Z 448.145,A -85,B 0,C 180,E1 -12852.258,E2 -12852.258} C_VEL
LIN {X 0,Y 369.04,Z 448.139,A -85,B 0,C 180,E1 -12856.228,E2 -12856.228} C_VEL
LIN {X 0,Y 369.07,Z 448.136,A -85,B 0,C 180,E1 -12860.132,E2 -12860.132} C_VEL
LIN {X 0,Y 369.177,Z 448.126,A -85,B 0,C 180,E1 -12863.441,E2 -12863.441} C_VEL
LIN {X 0,Y 369.322,Z 448.106,A -85,B 0,C 180,E1 -12867.819,E2 -12867.819} C_VEL
LIN {X 0,Y 369.461,Z 448.087,A -85,B 0,C 180,E1 -12870,E2 -12870} C_VEL
LIN {X 0,Y 369.321,Z 448.104,A -85,B 0,C 180,E1 -12872.181,E2 -12872.181} C_VEL
LIN {X 0,Y 369.2,Z 448.119,A -85,B 0,C 180,E1 -12876.558,E2 -12876.558} C_VEL
LIN {X 0,Y 369.071,Z 448.136,A -85,B 0,C 180,E1 -12879.868,E2 -12879.868} C_VEL
LIN {X 0,Y 369.04,Z 448.139,A -85,B 0,C 180,E1 -12883.772,E2 -12883.772} C_VEL
LIN {X 0,Y 369.004,Z 448.144,A -85,B 0,C 180,E1 -12887.768,E2 -12887.768} C_VEL
LIN {X 0,Y 368.931,Z 448.157,A -85,B 0,C 180,E1 -12891.219,E2 -12891.219} C_VEL
LIN {X 0,Y 368.96,Z 448.152,A -85,B 0,C 180,E1 -12894.775,E2 -12894.775} C_VEL
LIN {X 0,Y 368.964,Z 448.152,A -85,B 0,C 180,E1 -12897.203,E2 -12897.203} C_VEL
LIN {X 0,Y 368.92,Z 448.154,A -85,B 0,C 180,E1 -12899.689,E2 -12899.689} C_VEL
LIN {X 0,Y 368.883,Z 448.162,A -85,B 0,C 180,E1 -12903.039,E2 -12903.039} C_VEL
LIN {X 0,Y 368.844,Z 448.168,A -85,B 0,C 180,E1 -12904.982,E2 -12904.982} C_VEL
LIN {X 0,Y 368.378,Z 448.225,A -85,B 0,C 180,E1 -12908.536,E2 -12908.536} C_VEL
LIN {X 0,Y 368.159,Z 448.254,A -85,B 0,C 180,E1 -12910.469,E2 -12910.469} C_VEL
LIN {X 0,Y 368.009,Z 448.617,A -85,B 0,C 180,E1 -12911.943,E2 -12911.943} C_VEL
LIN {X 0,Y 367.945,Z 450.965,A -85,B 0,C 180,E1 -12914.721,E2 -12914.721} C_VEL
LIN {X 0,Y 367.281,Z 451.553,A -85,B 0,C 180,E1 -12915.323,E2 -12915.323} C_VEL
LIN {X 0,Y 364.401,Z 452.651,A -85,B 0,C 180,E1 -12916.26,E2 -12916.26} C_VEL
LIN {X 0,Y 361.476,Z 453.76,A -85,B 0,C 180,E1 -12917.211,E2 -12917.211} C_VEL
LIN {X 0,Y 360.773,Z 454.368,A -85,B 0,C 180,E1 -12917.829,E2 -12917.829} C_VEL
LIN {X 0,Y 360.78,Z 454.981,A -85,B 0,C 180,E1 -12918.523,E2 -12918.523} C_VEL
LIN {X 0,Y 365.501,Z 471.59,A -85,B 0,C 180,E1 -12919.46,E2 -12919.46} C_VEL
LIN {X 0,Y 368.96,Z 485.41,A -85,B 0,C 180,E1 -12920.43,E2 -12920.43} C_VEL
LIN {X 0,Y 369.644,Z 488.733,A -85,B 0,C 180,E1 -12920.691,E2 -12920.691} C_VEL
LIN {X 0,Y 368.459,Z 502.858,A -85,B 0,C 180,E1 -12921.735,E2 -12921.735} C_VEL
LIN {X 0,Y 367.286,Z 515.571,A -85,B 0,C 180,E1 -12922.932,E2 -12922.932} C_VEL
LIN {X 0,Y 365.994,Z 527.544,A -85,B 0,C 180,E1 -12924.318,E2 -12924.318} C_VEL
LIN {X 0,Y 364.724,Z 539.072,A -85,B 0,C 180,E1 -12925.952,E2 -12925.952} C_VEL
LIN {X 0,Y 363.68,Z 548.467,A -85,B 0,C 180,E1 -12927.568,E2 -12927.568} C_VEL
LIN {X 0,Y 362.603,Z 557.375,A -85,B 0,C 180,E1 -12929.417,E2 -12929.417} C_VEL
LIN {X 0,Y 361.928,Z 564.643,A -85,B 0,C 180,E1 -12931.275,E2 -12931.275} C_VEL
LIN {X 0,Y 361.275,Z 571.333,A -85,B 0,C 180,E1 -12933.421,E2 -12933.421} C_VEL
LIN {X 0,Y 360.874,Z 575.799,A -85,B 0,C 180,E1 -12935.246,E2 -12935.246} C_VEL
LIN {X 0,Y 360.598,Z 579.157,A -85,B 0,C 180,E1 -12937.058,E2 -12937.058} C_VEL
LIN {X 0,Y 360.403,Z 582.12,A -85,B 0,C 180,E1 -12939.39,E2 -12939.39} C_VEL
LIN {X 0,Y 360.337,Z 583.055,A -85,B 0,C 180,E1 -12940.636,E2 -12940.636} C_VEL
LIN {X 0,Y 360.332,Z 583.69,A -85,B 0,C 180,E1 -12942.988,E2 -12942.988} C_VEL
LIN {X 0,Y 360.506,Z 582.859,A -85,B 0,C 180,E1 -12945.319,E2 -12945.319} C_VEL
LIN {X 0,Y 360.852,Z 580.595,A -85,B 0,C 180,E1 -12947.629,E2 -12947.629} C_VEL
LIN {X 0,Y 361.403,Z 576.871,A -85,B 0,C 180,E1 -12949.92,E2 -12949.92} C_VEL
LIN {X 0,Y 362.019,Z 572.314,A -85,B 0,C 180,E1 -12951.916,E2 -12951.916} C_VEL
LIN {X 0,Y 362.926,Z 566.485,A -85,B 0,C 180,E1 -12953.886,E2 -12953.886} C_VEL
LIN {X 0,Y 364.097,Z 559.207,A -85,B 0,C 180,E1 -12955.849,E2 -12955.849} C_VEL
LIN {X 0,Y 365.436,Z 550.27,A -85,B 0,C 180,E1 -12957.795,E2 -12957.795} C_VEL
LIN {X 0,Y 366.967,Z 540.923,A -85,B 0,C 180,E1 -12959.451,E2 -12959.451} C_VEL
LIN {X 0,Y 368.673,Z 529.666,A -85,B 0,C 180,E1 -12961.092,E2 -12961.092} C_VEL
LIN {X 0,Y 370.281,Z 518.381,A -85,B 0,C 180,E1 -12962.447,E2 -12962.447} C_VEL
LIN {X 0,Y 371.89,Z 505.986,A -85,B 0,C 180,E1 -12963.657,E2 -12963.657} C_VEL
LIN {X 0,Y 373.301,Z 493.425,A -85,B 0,C 180,E1 -12964.642,E2 -12964.642} C_VEL
LIN {X 0,Y 371.706,Z 486.321,A -85,B 0,C 180,E1 -12965.315,E2 -12965.315} C_VEL
LIN {X 0,Y 367.617,Z 473.321,A -85,B 0,C 180,E1 -12966.533,E2 -12966.533} C_VEL
LIN {X 0,Y 362.911,Z 463.037,A -85,B 0,C 180,E1 -12967.531,E2 -12967.531} C_VEL
LIN {X 0,Y 361.913,Z 460.137,A -85,B 0,C 180,E1 -12967.782,E2 -12967.782} C_VEL
LIN {X 0,Y 362.017,Z 458.255,A -85,B 0,C 180,E1 -12971.194,E2 -12971.194} C_VEL
LIN {X 0,Y 362.202,Z 456.578,A -85,B 0,C 180,E1 -12974.61,E2 -12974.61} C_VEL
LIN {X 0,Y 362.481,Z 455.083,A -85,B 0,C 180,E1 -12978.19,E2 -12978.19} C_VEL
LIN {X 0,Y 362.579,Z 454.011,A -85,B 0,C 180,E1 -12981.61,E2 -12981.61} C_VEL
LIN {X 0,Y 362.571,Z 453.316,A -85,B 0,C 180,E1 -12985.242,E2 -12985.242} C_VEL
LIN {X 0,Y 362.562,Z 453.102,A -85,B 0,C 180,E1 -12987.725,E2 -12987.725} C_VEL
LIN {X 0,Y 362.59,Z 453.197,A -85,B 0,C 180,E1 -12990.262,E2 -12990.262} C_VEL
LIN {X 0,Y 362.692,Z 453.778,A -85,B 0,C 180,E1 -12993.57,E2 -12993.57} C_VEL
LIN {X 0,Y 362.894,Z 454.962,A -85,B 0,C 180,E1 -12996.896,E2 -12996.896} C_VEL
LIN {X 0,Y 363.201,Z 456.449,A -85,B 0,C 180,E1 -12999.684,E2 -12999.684} C_VEL
LIN {X 0,Y 363.593,Z 458.627,A -85,B 0,C 180,E1 -13002.735,E2 -13002.735} C_VEL
LIN {X 0,Y 364.07,Z 461.582,A -85,B 0,C 180,E1 -13005.978,E2 -13005.978} C_VEL
LIN {X 0,Y 364.551,Z 464.979,A -85,B 0,C 180,E1 -13009.046,E2 -13009.046} C_VEL
LIN {X 0,Y 364.605,Z 466.801,A -85,B 0,C 180,E1 -13010.5,E2 -13010.5} C_VEL
LIN {X 0,Y 364.167,Z 470.693,A -85,B 0,C 180,E1 -13013.255,E2 -13013.255} C_VEL
LIN {X 0,Y 363.421,Z 475.418,A -85,B 0,C 180,E1 -13016.259,E2 -13016.259} C_VEL
LIN {X 0,Y 362.662,Z 481.4,A -85,B 0,C 180,E1 -13019.745,E2 -13019.745} C_VEL
LIN {X 0,Y 361.904,Z 488.267,A -85,B 0,C 180,E1 -13023.472,E2 -13023.472} C_VEL
LIN {X 0,Y 361.807,Z 489.61,A -85,B 0,C 180,E1 -13024.172,E2 -13024.172} C_VEL
LIN {X 0,Y 362.786,Z 493.23,A -85,B 0,C 180,E1 -13024.41,E2 -13024.41} C_VEL
LIN {X 0,Y 366.718,Z 507.384,A -85,B 0,C 180,E1 -13025.447,E2 -13025.447} C_VEL
LIN {X 0,Y 369.034,Z 520.317,A -85,B 0,C 180,E1 -13026.427,E2 -13026.427} C_VEL
LIN {X 0,Y 370.138,Z 532.353,A -85,B 0,C 180,E1 -13027.4,E2 -13027.4} C_VEL
LIN {X 0,Y 370.369,Z 540.689,A -85,B 0,C 180,E1 -13028.137,E2 -13028.137} C_VEL
LIN {X 0,Y 368.488,Z 554.207,A -85,B 0,C 180,E1 -13029.372,E2 -13029.372} C_VEL
LIN {X 0,Y 366.895,Z 566.014,A -85,B 0,C 180,E1 -13030.706,E2 -13030.706} C_VEL
LIN {X 0,Y 365.402,Z 576.171,A -85,B 0,C 180,E1 -13032.077,E2 -13032.077} C_VEL
LIN {X 0,Y 363.916,Z 586.418,A -85,B 0,C 180,E1 -13033.739,E2 -13033.739} C_VEL
LIN {X 0,Y 362.764,Z 595.028,A -85,B 0,C 180,E1 -13035.413,E2 -13035.413} C_VEL
LIN {X 0,Y 361.836,Z 603.381,A -85,B 0,C 180,E1 -13037.379,E2 -13037.379} C_VEL
LIN {X 0,Y 361.054,Z 610.183,A -85,B 0,C 180,E1 -13039.344,E2 -13039.344} C_VEL
LIN {X 0,Y 360.622,Z 616.282,A -85,B 0,C 180,E1 -13041.595,E2 -13041.595} C_VEL
LIN {X 0,Y 360.456,Z 620.917,A -85,B 0,C 180,E1 -13043.919,E2 -13043.919} C_VEL
LIN {X 0,Y 360.414,Z 623.185,A -85,B 0,C 180,E1 -13045.527,E2 -13045.527} C_VEL
LIN {X 0,Y 360.484,Z 625.128,A -85,B 0,C 180,E1 -13047.765,E2 -13047.765} C_VEL
LIN {X 0,Y 360.529,Z 625.571,A -85,B 0,C 180,E1 -13048.883,E2 -13048.883} C_VEL
LIN {X 0,Y 360.536,Z 625.395,A -85,B 0,C 180,E1 -13051.117,E2 -13051.117} C_VEL
LIN {X 0,Y 360.533,Z 624.776,A -85,B 0,C 180,E1 -13052.234,E2 -13052.234} C_VEL
LIN {X 0,Y 360.436,Z 622.455,A -85,B 0,C 180,E1 -13054.473,E2 -13054.473} C_VEL
LIN {X 0,Y 360.508,Z 618.652,A -85,B 0,C 180,E1 -13056.717,E2 -13056.717} C_VEL
LIN {X 0,Y 360.636,Z 614.701,A -85,B 0,C 180,E1 -13058.404,E2 -13058.404} C_VEL
LIN {X 0,Y 360.901,Z 609.803,A -85,B 0,C 180,E1 -13060.094,E2 -13060.094} C_VEL
LIN {X 0,Y 361.531,Z 602.721,A -85,B 0,C 180,E1 -13062.062,E2 -13062.062} C_VEL
LIN {X 0,Y 362.077,Z 596.663,A -85,B 0,C 180,E1 -13063.469,E2 -13063.469} C_VEL
LIN {X 0,Y 362.924,Z 588.011,A -85,B 0,C 180,E1 -13065.154,E2 -13065.154} C_VEL
LIN {X 0,Y 364.114,Z 577.568,A -85,B 0,C 180,E1 -13066.829,E2 -13066.829} C_VEL
LIN {X 0,Y 365.374,Z 565.955,A -85,B 0,C 180,E1 -13068.359,E2 -13068.359} C_VEL
LIN {X 0,Y 366.678,Z 554.477,A -85,B 0,C 180,E1 -13069.598,E2 -13069.598} C_VEL
LIN {X 0,Y 367.93,Z 542.187,A -85,B 0,C 180,E1 -13070.681,E2 -13070.681} C_VEL
LIN {X 0,Y 368.253,Z 536.141,A -85,B 0,C 180,E1 -13071.143,E2 -13071.143} C_VEL
LIN {X 0,Y 366.441,Z 522.111,A -85,B 0,C 180,E1 -13072.155,E2 -13072.155} C_VEL
LIN {X 0,Y 363.916,Z 507.262,A -85,B 0,C 180,E1 -13073.017,E2 -13073.017} C_VEL
LIN {X 0,Y 361.511,Z 494.294,A -85,B 0,C 180,E1 -13073.609,E2 -13073.609} C_VEL
LIN {X 0,Y 362.035,Z 488.052,A -85,B 0,C 180,E1 -13076.751,E2 -13076.751} C_VEL
LIN {X 0,Y 362.771,Z 479.996,A -85,B 0,C 180,E1 -13080.889,E2 -13080.889} C_VEL
LIN {X 0,Y 363.424,Z 473.916,A -85,B 0,C 180,E1 -13084.111,E2 -13084.111} C_VEL
LIN {X 0,Y 364.192,Z 467.338,A -85,B 0,C 180,E1 -13087.702,E2 -13087.702} C_VEL
LIN {X 0,Y 364.292,Z 462.871,A -85,B 0,C 180,E1 -13090.262,E2 -13090.262} C_VEL
LIN {X 0,Y 363.428,Z 457.584,A -85,B 0,C 180,E1 -13093.508,E2 -13093.508} C_VEL
LIN {X 0,Y 362.38,Z 451.846,A -85,B 0,C 180,E1 -13097.251,E2 -13097.251} C_VEL
LIN {X 0,Y 361.922,Z 449.027,A -85,B 0,C 180,E1 -13099.228,E2 -13099.228} C_VEL
LIN {X 0,Y 361.863,Z 449.037,A -85,B 0,C 180,E1 -13102.982,E2 -13102.982} C_VEL
LIN {X 0,Y 361.858,Z 449.036,A -85,B 0,C 180,E1 -13106.629,E2 -13106.629} C_VEL
LIN {X 0,Y 361.872,Z 449.032,A -85,B 0,C 180,E1 -13109.672,E2 -13109.672} C_VEL
LIN {X 0,Y 361.95,Z 449.023,A -85,B 0,C 180,E1 -13113.475,E2 -13113.475} C_VEL
LIN {X 0,Y 361.885,Z 449.033,A -85,B 0,C 180,E1 -13117.144,E2 -13117.144} C_VEL
LIN {X 0,Y 361.901,Z 449.032,A -85,B 0,C 180,E1 -13120.723,E2 -13120.723} C_VEL
LIN {X 0,Y 361.927,Z 449.029,A -85,B 0,C 180,E1 -13123.066,E2 -13123.066} C_VEL
LIN {X 0,Y 361.993,Z 449.02,A -85,B 0,C 180,E1 -13126.528,E2 -13126.528} C_VEL
LIN {X 0,Y 362.026,Z 449.012,A -85,B 0,C 180,E1 -13129.938,E2 -13129.938} C_VEL
LIN {X 0,Y 362.145,Z 448.999,A -85,B 0,C 180,E1 -13132.193,E2 -13132.193} C_VEL
LIN {X 0,Y 362.113,Z 449.005,A -85,B 0,C 180,E1 -13134.431,E2 -13134.431} C_VEL
LIN {X 0,Y 362.278,Z 448.981,A -85,B 0,C 180,E1 -13137.777,E2 -13137.777} C_VEL
LIN {X 0,Y 362.422,Z 448.964,A -85,B 0,C 180,E1 -13140,E2 -13140} C_VEL
LIN {X 0,Y 362.278,Z 448.984,A -85,B 0,C 180,E1 -13142.224,E2 -13142.224} C_VEL
LIN {X 0,Y 362.172,Z 448.999,A -85,B 0,C 180,E1 -13146.686,E2 -13146.686} C_VEL
LIN {X 0,Y 362.069,Z 449.009,A -85,B 0,C 180,E1 -13148.934,E2 -13148.934} C_VEL
LIN {X 0,Y 361.955,Z 449.025,A -85,B 0,C 180,E1 -13152.333,E2 -13152.333} C_VEL
LIN {X 0,Y 361.957,Z 449.025,A -85,B 0,C 180,E1 -13154.621,E2 -13154.621} C_VEL
LIN {X 0,Y 361.955,Z 449.024,A -85,B 0,C 180,E1 -13158.1,E2 -13158.1} C_VEL
LIN {X 0,Y 361.887,Z 449.03,A -85,B 0,C 180,E1 -13161.654,E2 -13161.654} C_VEL
LIN {X 0,Y 361.924,Z 449.025,A -85,B 0,C 180,E1 -13165.291,E2 -13165.291} C_VEL
LIN {X 0,Y 361.91,Z 449.028,A -85,B 0,C 180,E1 -13167.779,E2 -13167.779} C_VEL
LIN {X 0,Y 361.843,Z 449.035,A -85,B 0,C 180,E1 -13171.286,E2 -13171.286} C_VEL
LIN {X 0,Y 361.851,Z 449.039,A -85,B 0,C 180,E1 -13174.281,E2 -13174.281} C_VEL
LIN {X 0,Y 361.862,Z 449.033,A -85,B 0,C 180,E1 -13177.224,E2 -13177.224} C_VEL
LIN {X 0,Y 361.833,Z 449.036,A -85,B 0,C 180,E1 -13180.756,E2 -13180.756} C_VEL
LIN {X 0,Y 361.817,Z 449.04,A -85,B 0,C 180,E1 -13184.369,E2 -13184.369} C_VEL
LIN {X 0,Y 361.856,Z 449.036,A -85,B 0,C 180,E1 -13187.565,E2 -13187.565} C_VEL
LIN {X 0,Y 361.874,Z 449.031,A -85,B 0,C 180,E1 -13190.973,E2 -13190.973} C_VEL
LIN {X 0,Y 361.875,Z 449.031,A -85,B 0,C 180,E1 -13194.656,E2 -13194.656} C_VEL
LIN {X 0,Y 361.839,Z 449.036,A -85,B 0,C 180,E1 -13198.371,E2 -13198.371} C_VEL
LIN {X 0,Y 361.904,Z 449.028,A -85,B 0,C 180,E1 -13200.956,E2 -13200.956} C_VEL
LIN {X 0,Y 361.957,Z 449.024,A -85,B 0,C 180,E1 -13203.476,E2 -13203.476} C_VEL
LIN {X 0,Y 361.893,Z 449.03,A -85,B 0,C 180,E1 -13207.145,E2 -13207.145} C_VEL
LIN {X 0,Y 361.924,Z 449.025,A -85,B 0,C 180,E1 -13210.725,E2 -13210.725} C_VEL
LIN {X 0,Y 361.949,Z 449.023,A -85,B 0,C 180,E1 -13214.227,E2 -13214.227} C_VEL
LIN {X 0,Y 362.002,Z 449.015,A -85,B 0,C 180,E1 -13216.528,E2 -13216.528} C_VEL
LIN {X 0,Y 362.034,Z 449.013,A -85,B 0,C 180,E1 -13219.938,E2 -13219.938} C_VEL
LIN {X 0,Y 362.139,Z 449.003,A -85,B 0,C 180,E1 -13223.313,E2 -13223.313} C_VEL
LIN {X 0,Y 362.286,Z 448.983,A -85,B 0,C 180,E1 -13227.777,E2 -13227.777} C_VEL
LIN {X 0,Y 362.43,Z 448.962,A -85,B 0,C 180,E1 -13230,E2 -13230} C_VEL
LIN {X 0,Y 362.285,Z 448.98,A -85,B 0,C 180,E1 -13232.223,E2 -13232.223} C_VEL
LIN {X 0,Y 362.162,Z 448.996,A -85,B 0,C 180,E1 -13236.686,E2 -13236.686} C_VEL
LIN {X 0,Y 362.035,Z 449.011,A -85,B 0,C 180,E1 -13240.062,E2 -13240.062} C_VEL
LIN {X 0,Y 362.001,Z 449.016,A -85,B 0,C 180,E1 -13243.899,E2 -13243.899} C_VEL
LIN {X 0,Y 361.97,Z 449.019,A -85,B 0,C 180,E1 -13247.938,E2 -13247.938} C_VEL
LIN {X 0,Y 361.894,Z 449.03,A -85,B 0,C 180,E1 -13251.652,E2 -13251.652} C_VEL
LIN {X 0,Y 361.93,Z 449.028,A -85,B 0,C 180,E1 -13255.289,E2 -13255.289} C_VEL
LIN {X 0,Y 361.916,Z 449.026,A -85,B 0,C 180,E1 -13257.778,E2 -13257.778} C_VEL
LIN {X 0,Y 361.846,Z 449.037,A -85,B 0,C 180,E1 -13261.284,E2 -13261.284} C_VEL
LIN {X 0,Y 361.788,Z 449.043,A -85,B 0,C 180,E1 -13264.287,E2 -13264.287} C_VEL
LIN {X 0,Y 361.504,Z 449.081,A -85,B 0,C 180,E1 -13267.147,E2 -13267.147} C_VEL
LIN {X 0,Y 361.084,Z 449.135,A -85,B 0,C 180,E1 -13270.616,E2 -13270.616} C_VEL
LIN {X 0,Y 360.985,Z 449.147,A -85,B 0,C 180,E1 -13271.447,E2 -13271.447} C_VEL
LIN {X 0,Y 360.865,Z 451.676,A -85,B 0,C 180,E1 -13274.698,E2 -13274.698} C_VEL
LIN {X 0,Y 360.773,Z 454.368,A -85,B 0,C 180,E1 -13277.829,E2 -13277.829} C_VEL
LIN {X 0,Y 361.221,Z 455.347,A -85,B 0,C 180,E1 -13278.238,E2 -13278.238} C_VEL
LIN {X 0,Y 362.607,Z 457.803,A -85,B 0,C 180,E1 -13278.652,E2 -13278.652} C_VEL
LIN {X 0,Y 364.526,Z 461.984,A -85,B 0,C 180,E1 -13278.992,E2 -13278.992} C_VEL
LIN {X 0,Y 365.148,Z 465.827,A -85,B 0,C 180,E1 -13279.177,E2 -13279.177} C_VEL
LIN {X 0,Y 364.323,Z 470.332,A -85,B 0,C 180,E1 -13279.325,E2 -13279.325} C_VEL
LIN {X 0,Y 361.383,Z 479.323,A -85,B 0,C 180,E1 -13279.645,E2 -13279.645} C_VEL
LIN {X 0,Y 361.257,Z 482.699,A -85,B 0,C 180,E1 -13279.847,E2 -13279.847} C_VEL
LIN {X 0,Y 361.351,Z 483.198,A -85,B 0,C 180,E1 -13279.883,E2 -13279.883} C_VEL
LIN {X 0,Y 362.732,Z 489.146,A -85,B 0,C 180,E1 -13280.356,E2 -13280.356} C_VEL
LIN {X 0,Y 361.782,Z 501.962,A -85,B 0,C 180,E1 -13281.321,E2 -13281.321} C_VEL
LIN {X 0,Y 360.604,Z 514.371,A -85,B 0,C 180,E1 -13282.479,E2 -13282.479} C_VEL
LIN {X 0,Y 359.239,Z 526.845,A -85,B 0,C 180,E1 -13283.915,E2 -13283.915} C_VEL
LIN {X 0,Y 358.104,Z 536.848,A -85,B 0,C 180,E1 -13285.309,E2 -13285.309} C_VEL
LIN {X 0,Y 357.016,Z 546.319,A -85,B 0,C 180,E1 -13286.888,E2 -13286.888} C_VEL
LIN {X 0,Y 355.832,Z 555.653,A -85,B 0,C 180,E1 -13288.771,E2 -13288.771} C_VEL
LIN {X 0,Y 355.068,Z 562.941,A -85,B 0,C 180,E1 -13290.563,E2 -13290.563} C_VEL
LIN {X 0,Y 354.537,Z 568.595,A -85,B 0,C 180,E1 -13292.235,E2 -13292.235} C_VEL
LIN {X 0,Y 354.043,Z 573.729,A -85,B 0,C 180,E1 -13294.105,E2 -13294.105} C_VEL
LIN {X 0,Y 353.646,Z 577.947,A -85,B 0,C 180,E1 -13296.084,E2 -13296.084} C_VEL
LIN {X 0,Y 353.414,Z 580.667,A -85,B 0,C 180,E1 -13297.8,E2 -13297.8} C_VEL
LIN {X 0,Y 353.319,Z 582.324,A -85,B 0,C 180,E1 -13299.208,E2 -13299.208} C_VEL
LIN {X 0,Y 353.226,Z 583.858,A -85,B 0,C 180,E1 -13301.437,E2 -13301.437} C_VEL
LIN {X 0,Y 353.265,Z 584.155,A -85,B 0,C 180,E1 -13302.73,E2 -13302.73} C_VEL
LIN {X 0,Y 353.391,Z 583.595,A -85,B 0,C 180,E1 -13305.017,E2 -13305.017} C_VEL
LIN {X 0,Y 353.736,Z 581.588,A -85,B 0,C 180,E1 -13307.376,E2 -13307.376} C_VEL
LIN {X 0,Y 354.296,Z 578.13,A -85,B 0,C 180,E1 -13309.716,E2 -13309.716} C_VEL
LIN {X 0,Y 355.014,Z 573.197,A -85,B 0,C 180,E1 -13312.034,E2 -13312.034} C_VEL
LIN {X 0,Y 355.833,Z 568.368,A -85,B 0,C 180,E1 -13313.763,E2 -13313.763} C_VEL
LIN {X 0,Y 356.983,Z 561.462,A -85,B 0,C 180,E1 -13315.766,E2 -13315.766} C_VEL
LIN {X 0,Y 358.4,Z 552.956,A -85,B 0,C 180,E1 -13317.752,E2 -13317.752} C_VEL
LIN {X 0,Y 359.949,Z 544.09,A -85,B 0,C 180,E1 -13319.44,E2 -13319.44} C_VEL
LIN {X 0,Y 361.721,Z 533.431,A -85,B 0,C 180,E1 -13321.113,E2 -13321.113} C_VEL
LIN {X 0,Y 363.535,Z 521.574,A -85,B 0,C 180,E1 -13322.631,E2 -13322.631} C_VEL
LIN {X 0,Y 365.347,Z 508.391,A -85,B 0,C 180,E1 -13323.998,E2 -13323.998} C_VEL
LIN {X 0,Y 366.927,Z 494.535,A -85,B 0,C 180,E1 -13325.145,E2 -13325.145} C_VEL
LIN {X 0,Y 363.803,Z 482.466,A -85,B 0,C 180,E1 -13326.367,E2 -13326.367} C_VEL
LIN {X 0,Y 360.415,Z 473.183,A -85,B 0,C 180,E1 -13327.298,E2 -13327.298} C_VEL
LIN {X 0,Y 356.157,Z 464.013,A -85,B 0,C 180,E1 -13328.259,E2 -13328.259} C_VEL
LIN {X 0,Y 354.902,Z 460.916,A -85,B 0,C 180,E1 -13328.542,E2 -13328.542} C_VEL
LIN {X 0,Y 355.02,Z 459.313,A -85,B 0,C 180,E1 -13331.418,E2 -13331.418} C_VEL
LIN {X 0,Y 355.229,Z 457.68,A -85,B 0,C 180,E1 -13334.904,E2 -13334.904} C_VEL
LIN {X 0,Y 355.527,Z 456.28,A -85,B 0,C 180,E1 -13338.438,E2 -13338.438} C_VEL
LIN {X 0,Y 355.623,Z 455.322,A -85,B 0,C 180,E1 -13341.748,E2 -13341.748} C_VEL
LIN {X 0,Y 355.632,Z 454.793,A -85,B 0,C 180,E1 -13344.628,E2 -13344.628} C_VEL
LIN {X 0,Y 355.63,Z 454.59,A -85,B 0,C 180,E1 -13348.313,E2 -13348.313} C_VEL
LIN {X 0,Y 355.697,Z 454.926,A -85,B 0,C 180,E1 -13351.832,E2 -13351.832} C_VEL
LIN {X 0,Y 355.806,Z 455.752,A -85,B 0,C 180,E1 -13354.947,E2 -13354.947} C_VEL
LIN {X 0,Y 356.056,Z 456.989,A -85,B 0,C 180,E1 -13357.859,E2 -13357.859} C_VEL
LIN {X 0,Y 356.367,Z 458.598,A -85,B 0,C 180,E1 -13360.602,E2 -13360.602} C_VEL
LIN {X 0,Y 356.763,Z 460.844,A -85,B 0,C 180,E1 -13363.589,E2 -13363.589} C_VEL
LIN {X 0,Y 357.226,Z 463.784,A -85,B 0,C 180,E1 -13366.713,E2 -13366.713} C_VEL
LIN {X 0,Y 357.595,Z 466.999,A -85,B 0,C 180,E1 -13369.567,E2 -13369.567} C_VEL
LIN {X 0,Y 357.373,Z 470.772,A -85,B 0,C 180,E1 -13372.438,E2 -13372.438} C_VEL
LIN {X 0,Y 356.501,Z 476.003,A -85,B 0,C 180,E1 -13375.892,E2 -13375.892} C_VEL
LIN {X 0,Y 355.626,Z 482.401,A -85,B 0,C 180,E1 -13379.74,E2 -13379.74} C_VEL
LIN {X 0,Y 354.88,Z 488.933,A -85,B 0,C 180,E1 -13383.371,E2 -13383.371} C_VEL
LIN {X 0,Y 355.818,Z 492.505,A -85,B 0,C 180,E1 -13383.641,E2 -13383.641} C_VEL
LIN {X 0,Y 359.431,Z 504.722,A -85,B 0,C 180,E1 -13384.602,E2 -13384.602} C_VEL
LIN {X 0,Y 361.933,Z 516.414,A -85,B 0,C 180,E1 -13385.535,E2 -13385.535} C_VEL
LIN {X 0,Y 363.501,Z 529.635,A -85,B 0,C 180,E1 -13386.645,E2 -13386.645} C_VEL
LIN {X 0,Y 363.84,Z 541.584,A -85,B 0,C 180,E1 -13387.724,E2 -13387.724} C_VEL
LIN {X 0,Y 361.834,Z 555.152,A -85,B 0,C 180,E1 -13389.02,E2 -13389.02} C_VEL
LIN {X 0,Y 360.049,Z 567.349,A -85,B 0,C 180,E1 -13390.472,E2 -13390.472} C_VEL
LIN {X 0,Y 358.34,Z 578.087,A -85,B 0,C 180,E1 -13392.007,E2 -13392.007} C_VEL
LIN {X 0,Y 356.861,Z 587.954,A -85,B 0,C 180,E1 -13393.702,E2 -13393.702} C_VEL
LIN {X 0,Y 355.546,Z 597.085,A -85,B 0,C 180,E1 -13395.597,E2 -13395.597} C_VEL
LIN {X 0,Y 354.602,Z 605.324,A -85,B 0,C 180,E1 -13397.699,E2 -13397.699} C_VEL
LIN {X 0,Y 353.872,Z 611.659,A -85,B 0,C 180,E1 -13399.704,E2 -13399.704} C_VEL
LIN {X 0,Y 353.497,Z 617.286,A -85,B 0,C 180,E1 -13402,E2 -13402} C_VEL
LIN {X 0,Y 353.33,Z 621.344,A -85,B 0,C 180,E1 -13404.292,E2 -13404.292} C_VEL
LIN {X 0,Y 353.301,Z 623.95,A -85,B 0,C 180,E1 -13406.579,E2 -13406.579} C_VEL
LIN {X 0,Y 353.464,Z 625.154,A -85,B 0,C 180,E1 -13408.861,E2 -13408.861} C_VEL
LIN {X 0,Y 353.473,Z 624.939,A -85,B 0,C 180,E1 -13411.139,E2 -13411.139} C_VEL
LIN {X 0,Y 353.435,Z 624.298,A -85,B 0,C 180,E1 -13412.279,E2 -13412.279} C_VEL
LIN {X 0,Y 353.368,Z 621.934,A -85,B 0,C 180,E1 -13414.563,E2 -13414.563} C_VEL
LIN {X 0,Y 353.426,Z 618.071,A -85,B 0,C 180,E1 -13416.852,E2 -13416.852} C_VEL
LIN {X 0,Y 353.581,Z 614.074,A -85,B 0,C 180,E1 -13418.573,E2 -13418.573} C_VEL
LIN {X 0,Y 353.843,Z 609.114,A -85,B 0,C 180,E1 -13420.297,E2 -13420.297} C_VEL
LIN {X 0,Y 354.496,Z 601.964,A -85,B 0,C 180,E1 -13422.305,E2 -13422.305} C_VEL
LIN {X 0,Y 355.287,Z 593.446,A -85,B 0,C 180,E1 -13424.239,E2 -13424.239} C_VEL
LIN {X 0,Y 356.37,Z 583.825,A -85,B 0,C 180,E1 -13426.027,E2 -13426.027} C_VEL
LIN {X 0,Y 357.519,Z 573.623,A -85,B 0,C 180,E1 -13427.592,E2 -13427.592} C_VEL
LIN {X 0,Y 358.956,Z 562.501,A -85,B 0,C 180,E1 -13428.996,E2 -13428.996} C_VEL
LIN {X 0,Y 360.108,Z 551.838,A -85,B 0,C 180,E1 -13430.119,E2 -13430.119} C_VEL
LIN {X 0,Y 361.45,Z 538.436,A -85,B 0,C 180,E1 -13431.263,E2 -13431.263} C_VEL
LIN {X 0,Y 359.904,Z 525.237,A -85,B 0,C 180,E1 -13432.276,E2 -13432.276} C_VEL
LIN {X 0,Y 357.423,Z 509.845,A -85,B 0,C 180,E1 -13433.241,E2 -13433.241} C_VEL
LIN {X 0,Y 354.627,Z 495.264,A -85,B 0,C 180,E1 -13433.942,E2 -13433.942} C_VEL
LIN {X 0,Y 354.493,Z 493.937,A -85,B 0,C 180,E1 -13434.01,E2 -13434.01} C_VEL
LIN {X 0,Y 355.101,Z 486.764,A -85,B 0,C 180,E1 -13437.716,E2 -13437.716} C_VEL
LIN {X 0,Y 355.704,Z 480.716,A -85,B 0,C 180,E1 -13440.91,E2 -13440.91} C_VEL
LIN {X 0,Y 356.37,Z 474.854,A -85,B 0,C 180,E1 -13444.077,E2 -13444.077} C_VEL
LIN {X 0,Y 357.11,Z 468.543,A -85,B 0,C 180,E1 -13447.595,E2 -13447.595} C_VEL
LIN {X 0,Y 357.303,Z 464.563,A -85,B 0,C 180,E1 -13449.905,E2 -13449.905} C_VEL
LIN {X 0,Y 356.855,Z 461.086,A -85,B 0,C 180,E1 -13452.036,E2 -13452.036} C_VEL
LIN {X 0,Y 355.925,Z 456.029,A -85,B 0,C 180,E1 -13455.303,E2 -13455.303} C_VEL
LIN {X 0,Y 354.953,Z 450.335,A -85,B 0,C 180,E1 -13459.202,E2 -13459.202} C_VEL
LIN {X 0,Y 354.872,Z 449.906,A -85,B 0,C 180,E1 -13459.565,E2 -13459.565} C_VEL
LIN {X 0,Y 354.794,Z 449.915,A -85,B 0,C 180,E1 -13463.54,E2 -13463.54} C_VEL
LIN {X 0,Y 354.826,Z 449.909,A -85,B 0,C 180,E1 -13466.317,E2 -13466.317} C_VEL
LIN {X 0,Y 354.85,Z 449.907,A -85,B 0,C 180,E1 -13470.321,E2 -13470.321} C_VEL
LIN {X 0,Y 354.894,Z 449.901,A -85,B 0,C 180,E1 -13474.172,E2 -13474.172} C_VEL
